# B&R Automation Studio project pneutrunk_plc (part 3)

#### Cyclic.st
```iecst
PROGRAM _CYCLIC

	TON_0(IN := kalibraciaStart, PT := T#5s0ms);

	IF buttons.klucik = FALSE THEN
		global_step		:= 0;
		step 			:= 7;
		buttons.stropBielaLED	:= FALSE;
	END_IF

	CASE step OF

		0:  // Detekcia referencnej polohy
			IF switch2 = FALSE THEN
				buttons.startLED				:= FALSE;
				switch2 						:= TRUE;
				FOR id:=0 TO 6 BY 1 DO
					modul.tlak1[id]	:= REAL_TO_INT(0);
					modul.tlak2[id]	:= REAL_TO_INT(0);
					modul.tlak3[id]	:= REAL_TO_INT(0);
					packetPos.qDesired[id*2] 	:= 0;
					packetPos.qDesired[id*2+1] 	:= 0;
					automatika.x_desired[id]	:= 0;
					automatika.y_desired[id]	:= 0;
					switch						:= FALSE;
				END_FOR

			END_IF

			IF buttons.startButton = TRUE THEN
				buttons.start	:= TRUE;
				global_step_udp	:= 0;
			END_IF

			IF buttons.start = TRUE AND buttons.centralStop = TRUE THEN
				buttons.stop					:= FALSE;
				buttons.stopLED					:= FALSE;
				buttons.stropCervenaLED			:= FALSE;
				buttons.startLED				:= TRUE;
				IF switch = FALSE THEN
					switch 						:= TRUE;
					kalibraciaStart 			:= TRUE;
					I_ON						:= TRUE;
					FOR id:=0 TO 6 BY 1 DO
						automatika.I_konstanta[id]	:= 25;
					END_FOR
					FOR id:=0 TO 6 BY 1 DO
						modul.tlak1[id]			:= REAL_TO_INT(3*32767/9);
						modul.tlak2[id]			:= REAL_TO_INT(3*32767/9);
						modul.tlak3[id]			:= REAL_TO_INT(3*32767/9);
					END_FOR
				END_IF

				IF switch = TRUE AND TON_0.Q = TRUE THEN
					switch			:= FALSE;
					kalibraciaStart	:= FALSE;
					step			:= 1;
				END_IF
			END_IF
			global_step				:= 0;
			buttons.stropBielaLED	:= TRUE;
		1:	// Vypustenie vzduchu zo vsetkych mechov, zapnutie I-regulatora
			(*
			FOR id:=0 TO 6 BY 1 DO
				modul.tlak1[id]	:= 0;
				modul.tlak2[id]	:= 0;
				modul.tlak3[id]	:= 0;
			END_FOR
			*)
			//I_ON					:= TRUE;
			switch2 				:= FALSE;
			kalibraciaStart			:= TRUE;

			step					:= 2;

		2:	// cakaj
			IF TON_0.Q = TRUE THEN
				kalibraciaStart		:= FALSE;
				step				:= 3;
			END_IF

		3:
			FOR id:=0 TO 6 BY 1 DO
				modull.nula_x[id]:= 0;
				modull.nula_y[id]:= 0;
			END_FOR

			step					:= 44;

			global_step 			:= 999;
			global_step_udp			:= 0;			// aby nahodou nemal na zaciatku gesto z predoslej udalosti

			kalibraciaStart			:= TRUE;
			(*
			FOR id:=0 TO 6 BY 1 DO
				modul.tlak1[id]	:= 0;
				modul.tlak2[id]	:= 0;
				modul.tlak3[id]	:= 0;
			END_FOR
			*)

		44:

			IF TON_0.Q = TRUE THEN
				kalibraciaStart		:= FALSE;
				step				:= 45;
				(*
				FOR id:=0 TO 6 BY 1 DO
					modull.nula_x[id]:= modul.uhol1[id]*1.0233 + 88.745;
					modull.nula_y[id]:= modul.uhol2[id];
				END_FOR
				*)
				modull.nula_x[0]:= modul.uhol1[0]*1.0233 + 88.745;
				modull.nula_x[1]:= modul.uhol1[1]*1.0228 + 88.871;
				modull.nula_x[2]:= modul.uhol1[2]*1.0235 + 90.761;
				modull.nula_x[3]:= modul.uhol1[3]*1.0254 + 88.307;
				modull.nula_x[4]:= modul.uhol1[4]*1.0216 + 90.3;
				modull.nula_x[5]:= modul.uhol1[5]*1.0039 + 87.274;
				modull.nula_x[6]:= modul.uhol1[6]*1.0065 + 87.623;

				modull.nula_y[0]:= modul.uhol2[0]*1.0275 + 89.292;
				modull.nula_y[1]:= modul.uhol2[1]*1.0079 + 89.873;
				modull.nula_y[2]:= modul.uhol2[2]*1.043 + 92.476;
				modull.nula_y[3]:= modul.uhol2[3]*1.0308 + 90.739;
				modull.nula_y[4]:= modul.uhol2[4]*1.008 + 86.877;
				modull.nula_y[5]:= modul.uhol2[5]*1.0009 + 87.856;
				modull.nula_y[6]:= modul.uhol2[6]*1.0258 + 90.567;
			END_IF
		45:
			kalibraciaStart		:= TRUE;
			step				:= 46;
		46:
			IF TON_0.Q = TRUE THEN
				kalibraciaStart	:= FALSE;
				step			:= 47;
			END_IF
		47:
			FOR id:=0 TO 6 BY 1 DO
				modul.tlak1[id]	:= 0;
				modul.tlak2[id]	:= 0;
				modul.tlak3[id]	:= 0;
			END_FOR
			step				:= 48;
			kalibraciaStart		:= TRUE;
		48:
			IF TON_0.Q = TRUE THEN
				kalibraciaStart	:= FALSE;
				step			:= 4;
			END_IF

		4:

			FOR id:=0 TO 6 BY 1 DO
			//	modull.real_uhol_x_kalibrovane[id]	:= modul.uhol1[id]*1.0233 + 88.745;
			//	modull.real_uhol_y_kalibrovane[id]	:= modul.uhol2[id];
			//	modul.uhol_XminusRef[id] 			:= modull.real_uhol_x_kalibrovane[id] - modull.nula_x[id];
			//	modul.uhol_YminusRef[id] 			:= modull.real_uhol_y_kalibrovane[id] - modull.nula_y[id];
				modul.linearReal		 			:= ref_linearny_posun;
			END_FOR

			modull.real_uhol_x_kalibrovane[0]:= modul.uhol1[0]*1.0233 + 88.745;
			modull.real_uhol_x_kalibrovane[1]:= modul.uhol1[1]*1.0228 + 88.871;
			modull.real_uhol_x_kalibrovane[2]:= modul.uhol1[2]*1.0235 + 90.761;
			modull.real_uhol_x_kalibrovane[3]:= modul.uhol1[3]*1.0254 + 88.307;
			modull.real_uhol_x_kalibrovane[4]:= modul.uhol1[4]*1.0216 + 90.3;
			modull.real_uhol_x_kalibrovane[5]:= modul.uhol1[5]*1.0039 + 87.274;
			modull.real_uhol_x_kalibrovane[6]:= modul.uhol1[6]*1.0065 + 87.623;

			modull.real_uhol_y_kalibrovane[0]:= modul.uhol2[0]*1.0275 + 89.292;
			modull.real_uhol_y_kalibrovane[1]:= modul.uhol2[1]*1.0079 + 89.873;
			modull.real_uhol_y_kalibrovane[2]:= modul.uhol2[2]*1.043 + 92.476;
			modull.real_uhol_y_kalibrovane[3]:= modul.uhol2[3]*1.0308 + 90.739;
			modull.real_uhol_y_kalibrovane[4]:= modul.uhol2[4]*1.008 + 86.877;
			modull.real_uhol_y_kalibrovane[5]:= modul.uhol2[5]*1.0009 + 87.856;
			modull.real_uhol_y_kalibrovane[6]:= modul.uhol2[6]*1.0258 + 90.567;

			IF (automatika.step_color = 1 OR automatika.step_color = 2) AND global_step = 0 THEN
				global_step			:= 999;
			END_IF

			zasobnik.ball			:= automatika.ball_up;
			zasobnik.ball_piston	:= automatika.ball_piston;
			zasobnik.ball_piston_sjf:= automatika.popcorn;
			zasobnik.levitovanie	:= automatika.levitacia;
			//modull.efektor			:= automatika.effector;
			I_konstanta_ID1			:= automatika.I_konstanta[0];
			I_konstanta_ID2			:= automatika.I_konstanta[1];
			I_konstanta_ID3			:= automatika.I_konstanta[2];
			I_konstanta_ID4			:= automatika.I_konstanta[3];
			I_konstanta_ID5			:= automatika.I_konstanta[4];
			I_konstanta_ID6			:= automatika.I_konstanta[5];
			I_konstanta_ID7			:= automatika.I_konstanta[6];

			IF buttons.stop = TRUE THEN
				buttons.start		:= FALSE;
				buttons.startLED	:= FALSE;
				buttons.stopLED		:= TRUE;
				global_step			:= 7;
			END_IF

			IF buttons.start = TRUE AND buttons.centralStop = TRUE THEN
				IF automatika.automatic = TRUE THEN
					IF automatika.holdPosition = FALSE THEN
						FOR id:=0 TO 6 BY 1 DO
							modull.pozadovany_uhol_y[id]	:=  packetPos.qDesired[id*2];
							modull.pozadovany_uhol_x[id]	:= -packetPos.qDesired[id*2+1];
						END_FOR
						modull.pozadovanyLinear				:= packetPos.qDesired[14]*7/25 + 23;
					END_IF
				ELSE
					FOR id:=0 TO 6 BY 1 DO
						modull.pozadovany_uhol_x[id]	:= automatika.x_desired[id];
						modull.pozadovany_uhol_y[id] 	:= automatika.y_desired[id];
					END_FOR
					modull.pozadovanyLinear				:= automatika.linear;
				END_IF

				// Joint limits
				FOR id:=0 TO 6 BY 1 DO
					IF modull.pozadovany_uhol_x[id] >= maxUhol THEN
						modull.pozadovany_uhol_x[id]	:= maxUhol;
					ELSIF modull.pozadovany_uhol_x[id] <= - maxUhol THEN
						modull.pozadovany_uhol_x[id] := -maxUhol;
					END_IF

					IF modull.pozadovany_uhol_y[id] >= maxUhol THEN
						modull.pozadovany_uhol_y[id]	:= maxUhol;
					ELSIF modull.pozadovany_uhol_y[id] <= - maxUhol THEN
						modull.pozadovany_uhol_y[id] := -maxUhol;
					END_IF

				END_FOR

				ref_alfa_x_ID1:= modull.pozadovany_uhol_x[0];
				ref_alfa_y_ID1:= modull.pozadovany_uhol_y[0];
				ref_alfa_x_ID2:= modull.pozadovany_uhol_x[1];
				ref_alfa_y_ID2:= modull.pozadovany_uhol_y[1];
				ref_alfa_x_ID3:= modull.pozadovany_uhol_x[2];
				ref_alfa_y_ID3:= modull.pozadovany_uhol_y[2];
				ref_alfa_x_ID4:= modull.pozadovany_uhol_x[3];
				ref_alfa_y_ID4:= modull.pozadovany_uhol_y[3];
				ref_alfa_x_ID5:= modull.pozadovany_uhol_x[4];
				ref_alfa_y_ID5:= modull.pozadovany_uhol_y[4];
				ref_alfa_x_ID6:= modull.pozadovany_uhol_x[5];
				ref_alfa_y_ID6:= modull.pozadovany_uhol_y[5];
				ref_alfa_x_ID7:= modull.pozadovany_uhol_x[6];
				ref_alfa_y_ID7:= modull.pozadovany_uhol_y[6];

				// Obmedzenie pre linearny posun (ak je hodnota nad 30 regulator sa sprava divne, nechce sa vypnut)
				IF modull.pozadovanyLinear >30 THEN
					ref_linearny_posun	:= 30;
				ELSIF modull.pozadovanyLinear <23 THEN
					ref_linearny_posun	:= 23;
				ELSE
					ref_linearny_posun	:= modull.pozadovanyLinear;
				END_IF

				(*
				act_alfa_x_ID1:= modull.real_uhol_x_kalibrovane[0] - modull.nula_x[0];
				act_alfa_y_ID1:= modull.real_uhol_y_kalibrovane[0] - modull.nula_y[0];
				act_alfa_x_ID2:= modull.real_uhol_x_kalibrovane[1] - modull.nula_x[1];
				act_alfa_y_ID2:= modull.real_uhol_y_kalibrovane[1] - modull.nula_y[1];
				act_alfa_x_ID3:= modull.real_uhol_x_kalibrovane[2] - modull.nula_x[2];
				act_alfa_y_ID3:= modull.real_uhol_y_kalibrovane[2] - modull.nula_y[2];
				act_alfa_x_ID4:= modull.real_uhol_x_kalibrovane[3] - modull.nula_x[3];
				act_alfa_y_ID4:= modull.real_uhol_y_kalibrovane[3] - modull.nula_y[3];
				act_alfa_x_ID5:= modull.real_uhol_x_kalibrovane[4] - modull.nula_x[4];
				act_alfa_y_ID5:= modull.real_uhol_y_kalibrovane[4] - modull.nula_y[4];
				act_alfa_x_ID6:= modull.real_uhol_x_kalibrovane[5] - modull.nula_x[5];
				act_alfa_y_ID6:= modull.real_uhol_y_kalibrovane[5] - modull.nula_y[5];
				act_alfa_x_ID7:= modull.real_uhol_x_kalibrovane[6] - modull.nula_x[6];
				act_alfa_y_ID7:= modull.real_uhol_y_kalibrovane[6] - modull.nula_y[6];
				*)
				(*
				act_alfa_x_ID1:= modull.real_uhol_x_kalibrovane[0] - modull.nula_x[0];
				act_alfa_y_ID1:= modull.real_uhol_y_kalibrovane[0] - modull.nula_y[0];
				act_alfa_x_ID2:= modull.real_uhol_x_kalibrovane[1] - modull.nula_x[1];
				act_alfa_y_ID2:= modull.real_uhol_y_kalibrovane[1] - modull.nula_y[1];
				act_alfa_x_ID3:= modull.real_uhol_x_kalibrovane[2] - modull.nula_x[2];
				act_alfa_y_ID3:= modull.real_uhol_y_kalibrovane[2] - modull.nula_y[2];
				act_alfa_x_ID4:= modull.real_uhol_x_kalibrovane[3] - modull.nula_x[3];
				act_alfa_y_ID4:= modull.real_uhol_y_kalibrovane[3] - modull.nula_y[3];
				act_alfa_x_ID5:= modull.real_uhol_x_kalibrovane[4] - modull.nula_x[4];
				act_alfa_y_ID5:= modull.real_uhol_y_kalibrovane[4] - modull.nula_y[4];
				act_alfa_x_ID6:= modull.real_uhol_x_kalibrovane[5] - modull.nula_x[5];
				act_alfa_y_ID6:= modull.real_uhol_y_kalibrovane[5] - modull.nula_y[5];
				act_alfa_x_ID7:= modull.real_uhol_x_kalibrovane[6] - modull.nula_x[6];
				act_alfa_y_ID7:= modull.real_uhol_y_kalibrovane[6] - modull.nula_y[6];
				*)
				// Pre experiment 2
				uhly.ref_alfa_x[0]	:= act_alfa_x_ID1;
				uhly.ref_alfa_y[0]	:= act_alfa_y_ID1;
				uhly.ref_alfa_x[1]	:= act_alfa_x_ID2;
				uhly.ref_alfa_y[1]	:= act_alfa_y_ID2;
				uhly.ref_alfa_x[2]	:= act_alfa_x_ID3;
				uhly.ref_alfa_y[2]	:= act_alfa_y_ID3;
				uhly.ref_alfa_x[3]	:= act_alfa_x_ID4;
				uhly.ref_alfa_y[3]	:= act_alfa_y_ID4;
				uhly.ref_alfa_x[4]	:= act_alfa_x_ID5;
				uhly.ref_alfa_y[4]	:= act_alfa_y_ID5;
				uhly.ref_alfa_x[5]	:= act_alfa_x_ID6;
				uhly.ref_alfa_y[5]	:= act_alfa_y_ID6;
				uhly.ref_alfa_x[6]	:= act_alfa_x_ID7;
				uhly.ref_alfa_y[6]	:= act_alfa_y_ID7;

				IF automatika.repeatability = FALSE THEN

					// Nastavenie tlakov podla regulacie
					// ID1
					id:=0;
					modul.tlak1[id] := REAL_TO_INT(Blue_tab_ID1*32767/9);
					modul.tlak2[id] := REAL_TO_INT(Green_tab_ID1*32767/9);
					modul.tlak3[id] := REAL_TO_INT(Yellow_tab_ID1*32767/9);

					// ID2
					id:=1;
					modul.tlak1[id] := REAL_TO_INT(Blue_tab_ID2*32767/9);
					modul.tlak2[id] := REAL_TO_INT(Green_tab_ID2*32767/9);
					modul.tlak3[id] := REAL_TO_INT(Yellow_tab_ID2*32767/9);

					// ID3
					id:=2;
					modul.tlak1[id] := REAL_TO_INT(Blue_tab_ID3*32767/9);
					modul.tlak2[id] := REAL_TO_INT(Green_tab_ID3*32767/9);
					modul.tlak3[id] := REAL_TO_INT(Yellow_tab_ID3*32767/9);

					// ID4
					id:=3;
					modul.tlak1[id] := REAL_TO_INT(Blue_tab_ID4*32767/9);
					modul.tlak2[id] := REAL_TO_INT(Green_tab_ID4*32767/9);
					modul.tlak3[id] := REAL_TO_INT(Yellow_tab_ID4*32767/9);

					// ID5
					id:=4;
					modul.tlak1[id] := REAL_TO_INT(Blue_tab_ID5*32767/9);
					modul.tlak2[id] := REAL_TO_INT(Green_tab_ID5*32767/9);
					modul.tlak3[id] := REAL_TO_INT(Yellow_tab_ID5*32767/9);

					// ID6
					id:=5;
					modul.tlak1[id] := REAL_TO_INT(Blue_tab_ID6*32767/9);
					modul.tlak2[id] := REAL_TO_INT(Green_tab_ID6*32767/9);
					modul.tlak3[id] := REAL_TO_INT(Yellow_tab_ID6*32767/9);

					// ID7
					id:=6;
					modul.tlak3[id] := REAL_TO_INT(Blue_tab_ID7*32767/9);
					modul.tlak1[id] := REAL_TO_INT(Green_tab_ID7*32767/9);
					modul.tlak2[id] := REAL_TO_INT(Yellow_tab_ID7*32767/9);

					//lin_modul
					modul.tlakLinear:= REAL_TO_INT(lin_pressure*32767/9);
				ELSE
					IF automatika.continuum = TRUE THEN

					ELSE

						FOR id:= 0 TO 5 BY 1 DO
							modul.tlak1[id] := automatika.desiredPressure1[id];
							modul.tlak2[id] := automatika.desiredPressure2[id];
							modul.tlak3[id] := automatika.desiredPressure3[id];
						END_FOR
						modul.tlakLinear	:= automatika.desiredPressureLinear;
					END_IF

				END_IF

			ELSIF buttons.centralStop = FALSE OR buttons.start = FALSE THEN
				buttons.start			:= FALSE;
				switch					:= FALSE;
				switch2					:= FALSE;
				I_ON					:= FALSE;
				kalibraciaStart			:= FALSE;
				step					:= 0;
				global_step_udp			:= 0;
				global_step				:= 0;
				step_repeatability		:= 0;
				automatika.repeatability:= FALSE;
				automatika.casovac		:= FALSE;
				automatika.ball_piston	:= FALSE;
				automatika.ball_up		:= FALSE;
				automatika.levitacia	:= FALSE;
				zasobnik.levitovanie	:= FALSE;
				zasobnik.ball_piston_sjf:= FALSE;
				automatika.popcorn		:= FALSE;
				automatika.casovac_uchopenie:= FALSE;
				automatika.effector		:= FALSE;
				automatika.holdPosition	:= FALSE;
				automatika.automatic	:= FALSE;
				act_alfa_x_ID1:= 0;
				act_alfa_y_ID1:= 0;
				act_alfa_x_ID2:= 0;
				act_alfa_y_ID2:= 0;
				act_alfa_x_ID3:= 0;
				act_alfa_y_ID3:= 0;
				act_alfa_x_ID4:= 0;
				act_alfa_y_ID4:= 0;
				act_alfa_x_ID5:= 0;
				act_alfa_y_ID5:= 0;
				act_alfa_x_ID6:= 0;
				act_alfa_y_ID6:= 0;
				act_alfa_x_ID7:= 0;
				act_alfa_y_ID7:= 0;
				ref_alfa_x_ID1:= 0;
				ref_alfa_y_ID1:= 0;
				ref_alfa_x_ID2:= 0;
				ref_alfa_y_ID2:= 0;
				ref_alfa_x_ID3:= 0;
				ref_alfa_y_ID3:= 0;
				ref_alfa_x_ID4:= 0;
				ref_alfa_y_ID4:= 0;
				ref_alfa_x_ID5:= 0;
				ref_alfa_y_ID5:= 0;
				ref_alfa_x_ID6:= 0;
				ref_alfa_y_ID6:= 0;
				ref_alfa_x_ID7:= 0;
				ref_alfa_y_ID7:= 0;
				FOR i:=0 TO 6 BY 1 DO
					modul.tlak1[i] 				:= 0;
					modul.tlak2[i]				:= 0;
					modul.tlak3[i] 				:= 0;
					modull.pozadovany_uhol_y[i]	:= 0;
					modull.pozadovany_uhol_x[i]	:= 0;
					modull.real_uhol_x_kalibrovane[i]	:= 0;
					modull.real_uhol_y_kalibrovane[i] 	:= 0;
					modull.nula_x[i]			:= 0;
					modull.nula_y[i]			:= 0;
				END_FOR
				modul.tlakLinear		:= 0;
			//	modull.efektor			:= FALSE;
				modull.pozadovanyLinear	:= 23;
				zasobnik.ball			:= FALSE;
				zasobnik.ball_piston	:= FALSE;
			END_IF
		5: // kolaborativny mod - doslo k narazu, alebo stlacenie stop
			buttons.startLED			:= FALSE;
			buttons.stopLED				:= TRUE;
			IF buttons.start = TRUE THEN
				buttons.stropBielaLED	:= FALSE;
				buttons.stropCervenaLED	:= TRUE;
				buttons.start			:= FALSE;
			END_IF
			step						:= 6;
			global_step					:= 0;

		6:
			IF buttons.stop = TRUE THEN
				buttons.stopLED			:= FALSE;
				buttons.stropCervenaLED	:= FALSE;
				buttons.stropBielaLED	:= TRUE;
				step					:= 7;
			END_IF

		7:	// resetovanie vsetkeho
			buttons.start			:= FALSE;
			switch					:= FALSE;
			switch2					:= FALSE;
			I_ON					:= FALSE;
			kalibraciaStart			:= FALSE;
			step					:= 0;
			global_step_udp			:= 0;
			global_step				:= 0;
			automatika.casovac		:= FALSE;
			zasobnik.levitovanie	:= FALSE;
			zasobnik.ball_piston_sjf:= FALSE;
			automatika.ball_piston	:= FALSE;
			automatika.ball_up		:= FALSE;
			automatika.popcorn		:= FALSE;
			zasobnik.ball_piston_sjf:= FALSE;
			automatika.casovac_uchopenie:= FALSE;
			automatika.effector		:= FALSE;
			automatika.holdPosition	:= FALSE;
			automatika.automatic	:= FALSE;
			act_alfa_x_ID1:= 0;
			act_alfa_y_ID1:= 0;
			act_alfa_x_ID2:= 0;
			act_alfa_y_ID2:= 0;
			act_alfa_x_ID3:= 0;
			act_alfa_y_ID3:= 0;
			act_alfa_x_ID4:= 0;
			act_alfa_y_ID4:= 0;
			act_alfa_x_ID5:= 0;
			act_alfa_y_ID5:= 0;
			act_alfa_x_ID6:= 0;
			act_alfa_y_ID6:= 0;
			act_alfa_x_ID7:= 0;
			act_alfa_y_ID7:= 0;
			ref_alfa_x_ID1:= 0;
			ref_alfa_y_ID1:= 0;
			ref_alfa_x_ID2:= 0;
			ref_alfa_y_ID2:= 0;
			ref_alfa_x_ID3:= 0;
			ref_alfa_y_ID3:= 0;
			ref_alfa_x_ID4:= 0;
			ref_alfa_y_ID4:= 0;
			ref_alfa_x_ID5:= 0;
			ref_alfa_y_ID5:= 0;
			ref_alfa_x_ID6:= 0;
			ref_alfa_y_ID6:= 0;
			ref_alfa_x_ID7:= 0;
			ref_alfa_y_ID7:= 0;
			FOR i:=0 TO 6 BY 1 DO
				modul.tlak1[i] 				:= 0;
				modul.tlak2[i]				:= 0;
				modul.tlak3[i] 				:= 0;
				modull.pozadovany_uhol_y[i]	:= 0;
				modull.pozadovany_uhol_x[i]	:= 0;
				modull.real_uhol_x_kalibrovane[i]	:= 0;
				modull.real_uhol_y_kalibrovane[i] 	:= 0;
				modull.nula_x[i]			:= 0;
				modull.nula_y[i]			:= 0;
			END_FOR
			modul.tlakLinear		:= 0;
		//	modull.efektor			:= FALSE;
			modull.pozadovanyLinear	:= 23;
			zasobnik.ball			:= FALSE;
			zasobnik.ball_piston	:= FALSE;
			IF buttons.klucik = FALSE THEN
				step				:= 8;
				global_step			:= 0;
			ELSE
				step				:= 0;
			END_IF
		8:
			IF buttons.klucik = TRUE THEN
				step				:= 0;
				global_step			:= 0;
			ELSE
				buttons.stropBielaLED	:= FALSE;
			END_IF

	END_CASE

	IF I_ON= TRUE THEN
		RESET_ID1:= TRUE;
		RESET_ID2:= TRUE;
		RESET_ID3:= TRUE;
		RESET_ID4:= TRUE;
		RESET_ID5:= TRUE;
		RESET_ID6:= TRUE;
		RESET_ID7:= TRUE;
	ELSE
		RESET_ID1:= FALSE;
		RESET_ID2:= FALSE;
		RESET_ID3:= FALSE;
		RESET_ID4:= FALSE;
		RESET_ID5:= FALSE;
		RESET_ID6:= FALSE;
		RESET_ID7:= FALSE;
	END_IF

	I_konstanta_ID1;
	I_konstanta_ID2;
	I_konstanta_ID3;
	I_konstanta_ID4;
	I_konstanta_ID5;
	I_konstanta_ID6;
	I_konstanta_ID7;

END_PROGRAM
```

#### Init.st
```iecst
PROGRAM _INIT
//	traj_0(ssMethodType := 2, aktualny_uhol_x := 0, aktualny_uhol_y := 0, pozadovany_uhol_x := 0, pozadovany_uhol_y :=0, dlzka_pohybu := 1);

//	traj_1(ssMethodType := 2, aktualny_uhol_x := 0, aktualny_uhol_y := 0, pozadovany_uhol_x := 0, pozadovany_uhol_y :=0, dlzka_pohybu := 1);

//	uhol2zdvyh_0(ssMethodType := 2, uhol_x := 15, uhol_y := 15);

	//FF_PID_r_t_0(ssMethodType := 0, ref_alfa_x := 0, ref_alfa_y := 0, real_alfa_x := 0, real_alfa_y := 0, P_parameter := 0, reset_PID_blue := 0, D_parameter := 0, N_parameter := 0, stiffness_ff := 3, reset_PID_green := 0, reset_PID_yellow := 0, tlak3 := 0, I_parameter := 0, tlak1 := 0, tlak2 := 0);
	FOR id:=0 TO 6 BY 1 DO
		modull.poradie[id]	:= 3;
	END_FOR

	maxUhol := 18;

	modull.FF_stiffness[0]	:= 3;
	stiffness_ff:= modull.FF_stiffness[0];
	switch := FALSE;
	poradie_ID1:=3;
	poradie_ID2:=3;
	poradie_ID3:=3;
	poradie_ID4:=3;
	poradie_ID5:=3;
	poradie_ID6:=3;
	poradie_ID7:=3;

	I_konstanta_ID1:=30;
	I_konstanta_ID2:=30;
	I_konstanta_ID3:=30;
	I_konstanta_ID4:=30;
	I_konstanta_ID5:=30;
	I_konstanta_ID6:=30;
	I_konstanta_ID7:=30;

	IF buttons.klucik = TRUE THEN
		buttons.stropBielaLED	:= TRUE;
	END_IF

	buttons.stropCervenaLED	:= FALSE;

END_PROGRAM
```

### Program Logical/Source/RS485/Sender (IEC) - sending serial data

#### SenderCyclic.st
```iecst
(********************************************************************
 * COPYRIGHT -- Bernecker + Rainer
 ********************************************************************
 * Program: Sender
 * File: SenderCyclic.st
 * Author: Bernecker & Rainer
 * Created: January 25, 2010
 ********************************************************************
 * Implementation of program Sender
 ********************************************************************)

(*************init program**********************)
PROGRAM _INIT
	Sender.Commands.open_send := TRUE;												(*enable sender by default*)
	packet485.sendPacketFinal[0] := 255;
	packet485.sendPacketFinal[1] := 255;
	packet485.sendPacketFinal[2] := 1;				// ID
	packet485.sendPacketFinal[3] := 1;
	packet485.sendPacketFinal[4] := 254;
	packet485.sendPacketFinal[5] := 254;
	Sender.step					 := FRM_WAIT;
END_PROGRAM

(*************cyclic program********************)
PROGRAM _CYCLIC

	CASE Sender.step OF
		FRM_WAIT:	(*--- wait for command*)

			IF Sender.Commands.open_send = TRUE THEN								(*command for sender activation*)
				Sender.step := FRM_OPEN;
   			END_IF

			(*close will be requested in step FRM_WRITE*)

		FRM_OPEN:	(*--- open serial interface*)

			(*Parameters for FRM_xopen()*)
			Sender.FRM_xopen_0.enable := TRUE;
			Sender.FRM_xopen_0.device := ADR('IF6.ST1.IF1');										(*Devicename --> see your serial interface properties*)
			Sender.FRM_xopen_0.mode := ADR('/PHY=RS485 /BD=38400 /DB=8 /PA=N /SB=1'); 		(*Modestring --> specifies the seria operation mode*)
			Sender.FRM_xopen_0.config := ADR(Sender.xopenConfig) ;					(*Additional Parameters, optional*)

			(*Additional Parameters for FRM_xopen()*)
			Sender.xopenConfig.idle := 10;											(*Idle time between two characters*)
			Sender.xopenConfig.delimc := 0;											(*activate two delimeters*)
			Sender.xopenConfig.delim[0] := 0; 										(*CR - carridge return -> dec 13*)
			Sender.xopenConfig.delim[1] := 0; 										(*LF - line feed -> dec 10*)
			Sender.xopenConfig.tx_cnt := 3;											(*number of transmit buffers*)
			Sender.xopenConfig.rx_cnt := 3; 										(*number of receive buffers*)
			Sender.xopenConfig.tx_len := 256; 										(*length of transmit buffers*)
			Sender.xopenConfig.rx_len := 256; 										(*lenght of receive buffers*)
			Sender.xopenConfig.argc := 0;											(*activate additional options*)
			Sender.xopenConfig.argv := 0;											(*parameters for additional options (check help)*)

			Sender.FRM_xopen_0();													(*call the FRM_xopen() function*)

			IF Sender.FRM_xopen_0.status = 0 THEN
				Sender.step := FRM_GBUF;											(*Interface opend successfully --> next step*)
			ELSIF Sender.FRM_xopen_0.status = BUSY THEN
				Sender.step := FRM_OPEN;											(*operation not finished yet --> call again*)
			ELSE
				Sender.step := FRM_ERROR;											(*function returned errorcode --> check help*)
   			END_IF

		FRM_GBUF:	(*--- aquire sendbuffer for FRM_WRITE*)
			Sender.FRM_gbuf_0.enable := TRUE;
   			Sender.FRM_gbuf_0.ident := Sender.FRM_xopen_0.ident;

			Sender.FRM_gbuf_0();													(*call the FRM_gbuf() function*)

			IF Sender.FRM_gbuf_0.status = 0 THEN
				memset(Sender.FRM_gbuf_0.buffer,0,Sender.FRM_gbuf_0.buflng);		(*clear sendbuffer*)
				Sender.step := FRM_PREPARE_SENDDATA;								(*system returned a valid buffer --> next step*)
			ELSIF Sender.FRM_gbuf_0.status = BUSY THEN
				Sender.step := FRM_GBUF;											(*operation not finished yet --> call again*)
			ELSE
				Sender.step := FRM_ERROR;											(*function returned errorcode --> check help*)
   			END_IF

		FRM_PREPARE_SENDDATA: (*--- prepare senddata, copy data to sendbuffer*)

			IF packet485.id = 8 THEN
				packet485.id := 1;
			ELSE
				packet485.id := packet485.id + 1;
			END_IF
			Sender.Commands.open_send := TRUE;										(*enable sender by default*)
			packet485.sendPacketFinal[0] := 255;
			packet485.sendPacketFinal[1] := 255;
			packet485.sendPacketFinal[2] := USINT_TO_BYTE(packet485.id);
			packet485.sendPacketFinal[3] := 1;
			packet485.sendPacketFinal[4] := 254;
			packet485.sendPacketFinal[5] := 254;
			packet485.sendPacketFinal[0] := 255;

			strcpy(Sender.FRM_gbuf_0.buffer,ADR(packet485.sendPacketFinal));		(*copy senddata to sendbuffer*)
			Sender.step := FRM_WRITE;												(*--> next step*)

		FRM_WRITE:	(*--- write data to interface*)

			(*Parameters for FRM_write()*)
			Sender.FRM_write_0.enable := TRUE;
			Sender.FRM_write_0.ident := Sender.FRM_xopen_0.ident;					(*ident from FRM_xopen()*)
			Sender.FRM_write_0.buffer := Sender.FRM_gbuf_0.buffer;					(*sendbuffer*)
			Sender.FRM_write_0.buflng := strlen(ADR(packet485.sendPacketFinal));				(*net length of senddata*)

			Sender.FRM_write_0();													(*call the FRM_write() function*)

			IF Sender.FRM_write_0.status = 0 THEN
				IF Sender.Commands.close = TRUE THEN								(*requst to close the serial port*)
					Sender.Commands.open_send := FALSE;								(*disable command open_send*)
					Sender.step := FRM_CLOSE;
				ELSE
					Sender.step := FRM_GBUF;										(*writing successful --> get next sendbuffer*)
				END_IF
			ELSIF Sender.FRM_write_0.status = BUSY THEN
				Sender.step := FRM_WRITE;											(*operation not finished yet --> call again*)
			ELSE
				Sender.step := FRM_ROBUF;											(*function returned errorcode --> check help*)
   			END_IF

		FRM_ROBUF:	(*--- release sendbuffer in case of no successful write operation*)
			Sender.FRM_robuf_0.enable := TRUE;
			Sender.FRM_robuf_0.buffer := Sender.FRM_gbuf_0.buffer;					(*sendbuffer*)
			Sender.FRM_robuf_0.buflng := Sender.FRM_gbuf_0.buflng;					(*buffer length*)
			Sender.FRM_robuf_0.ident := Sender.FRM_xopen_0.ident;					(*ident open*)

			Sender.FRM_robuf_0();													(*call the FRM_robuf() function*)

			IF Sender.FRM_robuf_0.status = 0 THEN
				Sender.step := FRM_GBUF;											(*released buffer successful --> get next sendbuffer*)
			ELSIF Sender.FRM_robuf_0.status = BUSY THEN
				Sender.step := FRM_ROBUF;											(*operation not finished yet --> call again*)
			ELSE
				Sender.step := FRM_ERROR;											(*function returned errorcode --> check help*)
   			END_IF

		FRM_CLOSE:	(*--- close the interface*)
			Sender.FRM_close_0.enable := TRUE;
   			Sender.FRM_close_0.ident := Sender.FRM_xopen_0.ident;					(*ident from FRM_xopen()*)

			Sender.FRM_close_0();													(*call the FRM_close() function*)

			IF Sender.FRM_close_0.status = 0 THEN
				Sender.Commands.close := FALSE;										(*disable close command*)
				Sender.step := FRM_WAIT;											(*closed interface successfully --> wait step*)
			ELSIF Sender.FRM_close_0.status = BUSY THEN
				Sender.step := FRM_CLOSE;											(*operation not finished yet --> call again*)
			ELSE
				Sender.step := FRM_ERROR;											(*function returned errorcode --> check help*)
			END_IF

		FRM_ERROR:	(*--- error handling*)
			Sender.step := FRM_WAIT;
			//; (*not implementet yet, check help for error codes*)
 	END_CASE

END_PROGRAM
```

### Program Logical/Source/RS485/Receiver (IEC) - receiving serial data

#### ReceiverCyclic.st
```iecst
(********************************************************************
 * COPYRIGHT -- Bernecker + Rainer
 ********************************************************************
 * Program: Receiver
 * File: ReceiverCyclic.st
 * Author: Bernecker & Rainer
 * Created: January 25, 2010
 ********************************************************************
 * Implementation of program Receiver
 ********************************************************************)

(*************init program**********************)
PROGRAM _INIT
	Receiver.Commands.open_receive := TRUE;												(*enable Receiver by default*)
END_PROGRAM

(*************cyclic program********************)
PROGRAM _CYCLIC

	CASE Receiver.step OF
		FRM_WAIT:	(*--- wait for command*)

			IF Receiver.Commands.open_receive = TRUE THEN								(*command for Receiver activation*)
				Receiver.step := FRM_OPEN;
   			END_IF

			(*close will be requested in step FRM_RBUF*)

		FRM_OPEN:	(*--- open serial interface*)

			(*Parameters for FRM_xopen()*)
			Receiver.FRM_xopen_0.enable := TRUE;
			Receiver.FRM_xopen_0.device := ADR('IF6.ST1.IF1');							(*Devicename --> see your serial interface properties*)
			Receiver.FRM_xopen_0.mode := ADR('/PHY=RS485 /BD=38400 /DB=8 /PA=N /SB=1'); (*Modestring --> specifies the seria operation mode*)
			Receiver.FRM_xopen_0.config := ADR(Receiver.xopenConfig) ;					(*Additional Parameters, optional*)

			(*Additional Parameters for FRM_xopen()*)
			Receiver.xopenConfig.idle := 10;											(*Idle time between two characters*)
			Receiver.xopenConfig.delimc := 0;											(*activate two delimeters*)
			Receiver.xopenConfig.delim[0] := 0; 										(*e.g. CR - carridge return -> dec 13*)
			Receiver.xopenConfig.delim[1] := 0; 										(*e.g. LF - line feed -> dec 10*)
			Receiver.xopenConfig.tx_cnt := 3;											(*number of transmit buffers*)
			Receiver.xopenConfig.rx_cnt := 3; 											(*number of receive buffers*)
			Receiver.xopenConfig.tx_len := 256; 										(*length of transmit buffers*)
			Receiver.xopenConfig.rx_len := 256; 										(*lenght of receive buffers*)
			Receiver.xopenConfig.argc := 0;												(*activate additional options*)
			Receiver.xopenConfig.argv := 0;												(*parameters for additional options (check help)*)

			Receiver.FRM_xopen_0();														(*call the FRM_xopen() function*)

			IF Receiver.FRM_xopen_0.status = 0 THEN
				Receiver.step := FRM_READ;												(*Interface opend successfully --> next step*)
			ELSIF Receiver.FRM_xopen_0.status = BUSY THEN
				Receiver.step := FRM_OPEN;												(*operation not finished yet --> call again*)
			ELSE
				Receiver.step := FRM_ERROR;												(*function returned errorcode --> check help*)
   			END_IF

		FRM_READ:	(*--- read data from serial interface*)
			Receiver.FRM_read_0.enable := TRUE;
   			Receiver.FRM_read_0.ident := Receiver.FRM_xopen_0.ident;

			Receiver.FRM_read_0();														(*call the FRM_read() function*)

			IF Receiver.FRM_read_0.status = 0 THEN
				Receiver.step := FRM_COPY_RD_DATA;										(*system returned a valid data --> next step*)
			ELSIF Receiver.FRM_read_0.status = frmERR_NOINPUT THEN
				Receiver.step := FRM_READ;												(*no data available --> call again*)
			ELSIF Receiver.FRM_read_0.status = frmERR_INPUTERROR THEN
				Receiver.step := FRM_RBUF;												(*received Frame with defective characters, skip data*)
			ELSE
				Receiver.step := FRM_ERROR;												(*function returned errorcode --> check help*)
   			END_IF

		FRM_COPY_RD_DATA: (*--- copy data out of the receive buffer*)
			(*
			FOR i:=0 TO 8 BY 1 DO
				packet485.packet[i] := Receiver.receive_data[i];
			END_FOR
			*)
			memset(ADR(Receiver.receive_data),0,SIZEOF(Receiver.receive_data));			(*clear read_data buffer*)
			memcpy(ADR(Receiver.receive_data),Receiver.FRM_read_0.buffer,Receiver.FRM_read_0.buflng);     (*copy and evaluate read data*)

			IF(Receiver.receive_data[0] = 255)THEN
				IF(Receiver.receive_data[1] = 255)THEN
					IF(Receiver.receive_data[9] = 254)THEN
						IF(Receiver.receive_data[10] = 254)THEN
							IF(Receiver.receive_data[2] = 1)THEN
								modul.uholINT1 := BYTE_TO_INT(Receiver.receive_data[5]);
								modul.uholINT1 := SHL(modul.uholINT1,8);
								modul.uholINT1  := modul.uholINT1  + BYTE_TO_INT(Receiver.receive_data[6]);
								modul.uhol1[0] := INT_TO_REAL(modul.uholINT1);
								modul.uhol1[0] := modul.uhol1[0]*260/1024 - 130;
								modul.uholINT2 := BYTE_TO_INT(Receiver.receive_data[7]);
								modul.uholINT2 := SHL(modul.uholINT2,8);
								modul.uholINT2  := modul.uholINT2  + BYTE_TO_INT(Receiver.receive_data[8]);
								modul.uhol2[0] := INT_TO_REAL(modul.uholINT2);
								modul.uhol2[0] := modul.uhol2[0]*260/1024 - 130;
							ELSIF(Receiver.receive_data[2] = 2)THEN
								modul.uholINT1 := BYTE_TO_INT(Receiver.receive_data[5]);
								modul.uholINT1 := SHL(modul.uholINT1,8);
								modul.uholINT1  := modul.uholINT1  + BYTE_TO_INT(Receiver.receive_data[6]);
								modul.uhol1[1] := INT_TO_REAL(modul.uholINT1);
								modul.uhol1[1] := modul.uhol1[1]*260/1024 - 130;
								modul.uholINT2 := BYTE_TO_INT(Receiver.receive_data[7]);
								modul.uholINT2 := SHL(modul.uholINT2,8);
								modul.uholINT2  := modul.uholINT2  + BYTE_TO_INT(Receiver.receive_data[8]);
								modul.uhol2[1] := INT_TO_REAL(modul.uholINT2);
								modul.uhol2[1] := modul.uhol2[1]*260/1024 - 130;
							ELSIF(Receiver.receive_data[2] = 3)THEN
								modul.uholINT1 := BYTE_TO_INT(Receiver.receive_data[5]);
								modul.uholINT1 := SHL(modul.uholINT1,8);
								modul.uholINT1  := modul.uholINT1  + BYTE_TO_INT(Receiver.receive_data[6]);
								modul.uhol1[2] := INT_TO_REAL(modul.uholINT1);
								modul.uhol1[2] := modul.uhol1[2]*260/1024 - 130;
								modul.uholINT2 := BYTE_TO_INT(Receiver.receive_data[7]);
								modul.uholINT2 := SHL(modul.uholINT2,8);
								modul.uholINT2  := modul.uholINT2  + BYTE_TO_INT(Receiver.receive_data[8]);
								modul.uhol2[2] := INT_TO_REAL(modul.uholINT2);
								modul.uhol2[2] := modul.uhol2[2]*260/1024 - 130;
								IF Receiver.receive_data[4] = 3 OR Receiver.receive_data[4] > 15 THEN
									modul.naraz[2]	:= TRUE;
								ELSE
									modul.naraz[2]	:= FALSE;
								END_IF
							ELSIF(Receiver.receive_data[2] = 4)THEN
								modul.uholINT1 := BYTE_TO_INT(Receiver.receive_data[5]);
								modul.uholINT1 := SHL(modul.uholINT1,8);
								modul.uholINT1  := modul.uholINT1  + BYTE_TO_INT(Receiver.receive_data[6]);
								modul.uhol1[3] := INT_TO_REAL(modul.uholINT1);
								modul.uhol1[3] := modul.uhol1[3]*260/1024 - 130;
								modul.uholINT2 := BYTE_TO_INT(Receiver.receive_data[7]);
								modul.uholINT2 := SHL(modul.uholINT2,8);
								modul.uholINT2  := modul.uholINT2  + BYTE_TO_INT(Receiver.receive_data[8]);
								modul.uhol2[3] := INT_TO_REAL(modul.uholINT2);
								modul.uhol2[3] := modul.uhol2[3]*260/1024 - 130;
								IF Receiver.receive_data[4] = 3 OR Receiver.receive_data[4] > 15 THEN
									modul.naraz[3]	:= TRUE;
								ELSE
									modul.naraz[3]	:= FALSE;
								END_IF
							ELSIF(Receiver.receive_data[2] = 5)THEN
								modul.uholINT1 := BYTE_TO_INT(Receiver.receive_data[5]);
								modul.uholINT1 := SHL(modul.uholINT1,8);
								modul.uholINT1  := modul.uholINT1  + BYTE_TO_INT(Receiver.receive_data[6]);
								modul.uhol1[4] := INT_TO_REAL(modul.uholINT1);
								modul.uhol1[4] := modul.uhol1[4]*260/1024 - 130;
								modul.uholINT2 := BYTE_TO_INT(Receiver.receive_data[7]);
								modul.uholINT2 := SHL(modul.uholINT2,8);
								modul.uholINT2  := modul.uholINT2  + BYTE_TO_INT(Receiver.receive_data[8]);
								modul.uhol2[4] := INT_TO_REAL(modul.uholINT2);
								modul.uhol2[4] := modul.uhol2[4]*260/1024 - 130;
								IF Receiver.receive_data[4] = 3 OR Receiver.receive_data[4] > 15  THEN
									modul.naraz[4]	:= TRUE;
								ELSE
									modul.naraz[4]	:= FALSE;
								END_IF
							ELSIF(Receiver.receive_data[2] = 6)THEN
								modul.uholINT1 := BYTE_TO_INT(Receiver.receive_data[5]);
								modul.uholINT1 := SHL(modul.uholINT1,8);
								modul.uholINT1  := modul.uholINT1  + BYTE_TO_INT(Receiver.receive_data[6]);
								modul.uhol1[5] := INT_TO_REAL(modul.uholINT1);
								modul.uhol1[5] := modul.uhol1[5]*260/1024 - 130;
								modul.uholINT2 := BYTE_TO_INT(Receiver.receive_data[7]);
								modul.uholINT2 := SHL(modul.uholINT2,8);
								modul.uholINT2  := modul.uholINT2  + BYTE_TO_INT(Receiver.receive_data[8]);
								modul.uhol2[5] := INT_TO_REAL(modul.uholINT2);
								modul.uhol2[5] := modul.uhol2[5]*260/1024 - 130;
								IF Receiver.receive_data[4] = 3 OR Receiver.receive_data[4] > 15 THEN
									modul.naraz[5]	:= TRUE;
								ELSE
									modul.naraz[5]	:= FALSE;
								END_IF
							ELSIF(Receiver.receive_data[2] = 7)THEN
								modul.uholINT1 := BYTE_TO_INT(Receiver.receive_data[5]);
								modul.uholINT1 := SHL(modul.uholINT1,8);
								modul.uholINT1  := modul.uholINT1  + BYTE_TO_INT(Receiver.receive_data[6]);
								modul.uhol1[6] := INT_TO_REAL(modul.uholINT1);
								modul.uhol1[6] := modul.uhol1[6]*260/1024 - 130;
								modul.uholINT2 := BYTE_TO_INT(Receiver.receive_data[7]);
								modul.uholINT2 := SHL(modul.uholINT2,8);
								modul.uholINT2  := modul.uholINT2  + BYTE_TO_INT(Receiver.receive_data[8]);
								modul.uhol2[6] := INT_TO_REAL(modul.uholINT2);
								modul.uhol2[6] := modul.uhol2[6]*260/1024 - 130;
								IF Receiver.receive_data[4] = 1 OR Receiver.receive_data[4] = 2 OR Receiver.receive_data[4] > 15  THEN //lebo dve moduly su zapojene do jednej dosky
									modul.naraz[6]	:= TRUE;
								ELSE
									modul.naraz[6]	:= FALSE;
								END_IF
							ELSIF(Receiver.receive_data[2] = 8)THEN
								IF Receiver.receive_data[4] = 3 OR Receiver.receive_data[4] > 15 THEN
									modul.naraz[7]	:= TRUE;
								ELSE
									modul.naraz[7]	:= FALSE;
								END_IF
							END_IF
						END_IF
					END_IF
				END_IF
			END_IF

			Receiver.step := FRM_RBUF;													(*release read buffer*)

		FRM_RBUF:	(*--- release readbuffer*)

			(*Parameters for FRM_rbuf()*)
			Receiver.FRM_rbuf_0.enable := TRUE;
			Receiver.FRM_rbuf_0.ident := Receiver.FRM_xopen_0.ident;					(*ident from FRM_xopen()*)
			Receiver.FRM_rbuf_0.buffer := Receiver.FRM_read_0.buffer;					(*read buffer*)
			Receiver.FRM_rbuf_0.buflng := Receiver.FRM_read_0.buflng;					(*length of sendbuffer*)

			Receiver.FRM_rbuf_0();														(*call the FRM_rbuf() function*)

			IF Receiver.FRM_rbuf_0.status = 0 THEN
				IF Receiver.Commands.close = TRUE THEN
					Receiver.Commands.open_receive := FALSE;								(*disable command open_send*)
					Receiver.step := FRM_CLOSE;											(*request to close serial port*)
				ELSE
					Receiver.step := FRM_READ;											(*read again*)
				END_IF
			ELSIF Receiver.FRM_rbuf_0.status = BUSY THEN
				Receiver.step := FRM_RBUF;												(*operation not finished yet --> call again*)
			ELSIF Receiver.FRM_rbuf_0.status = frmERR_INVALIDBUFFER THEN
				Receiver.step := FRM_READ;												(*buffer is invalid --> read again*)
			ELSE
				Receiver.step := FRM_ERROR;												(*function returned errorcode --> check help*)
   			END_IF

		FRM_CLOSE:	(*--- close the interface*)
			Receiver.FRM_close_0.enable := TRUE;
   			Receiver.FRM_close_0.ident := Receiver.FRM_xopen_0.ident;					(*ident from FRM_xopen()*)

			Receiver.FRM_close_0();														(*call the FRM_close() function*)

			IF Receiver.FRM_close_0.status = 0 THEN
				Receiver.Commands.close := FALSE;										(*disable close command*)
				Receiver.step := FRM_WAIT;												(*closed interface successfully --> wait step*)
			ELSIF Receiver.FRM_close_0.status = BUSY THEN
				Receiver.step := FRM_CLOSE;												(*operation not finished yet --> call again*)
			ELSE
				Receiver.step := FRM_ERROR;												(*function returned errorcode --> check help*)
			END_IF

		FRM_ERROR:	(*--- error handling*)
			; (*not implementet yet, check help for error codes*)
 	END_CASE

END_PROGRAM
```

### Program Logical/Source/Testing (IEC)

#### Cyclic.st
```iecst
PROGRAM _CYCLIC

	IF i >= 30000 THEN
		i := 0;
	ELSE
		i := i + 100;
	END_IF

	modul.tlak1[0] := i;

END_PROGRAM
```

### Program Logical/Source/Experiments/Continuum

#### Variables.var
```iecst
VAR
	pressure : tlak;
	id : INT;
END_VAR
```

#### Cyclic.st
```iecst
PROGRAM _CYCLIC
	automatika.continuum	:= TRUE;
	FOR id:=0 TO 5 BY 1 DO
		modul.tlak1[id]	:= REAL_TO_INT(pressure.p1*32767/9);
		modul.tlak2[id]	:= REAL_TO_INT(pressure.p2*32767/9);
		modul.tlak3[id]	:= REAL_TO_INT(pressure.p3*32767/9);
	END_FOR
	modul.tlak2[6]	:= REAL_TO_INT(pressure.p3*32767/9);
	modul.tlak3[6]	:= REAL_TO_INT(pressure.p2*32767/9);
	modul.tlak1[6]	:= REAL_TO_INT(pressure.p1*32767/9);

END_PROGRAM
```

### Program Logical/Source/Experiments/HandControl

#### Cyclic.st
```iecst
PROGRAM _CYCLIC

	FOR id:=0 TO 6 BY 1 DO
		automatika.x_desired[id]	:= (uhly.ref_alfa_x[id]);
		automatika.y_desired[id]	:= (uhly.ref_alfa_y[id]);
	END_FOR

END_PROGRAM
```

### Program Logical/Source/Experiments/Repeatability

#### Variables.var
```iecst
VAR
	casovac_start : BOOL;
	TON_0 : TON;
	i : INT;
	TON_1 : TON;
	pauza : BOOL;
	TON_2 : TON;
	kameraBool : BOOL;
END_VAR
```

#### Cyclic.st
```iecst
PROGRAM _CYCLIC

	TON_0(IN := casovac_start, PT := INT_TO_TIME(automatika.cas));
	TON_1(IN := pauza, PT := T#10s0ms);
	TON_2(IN := kameraBool, PT := T#1s0ms);

	IF step = 4 THEN

		CASE automatika.step_repeatability OF
			0:
				casovac_start					:= TRUE;
				automatika.step_repeatability	:= 1;
				automatika.repeatability		:= TRUE;
				automatika.cas					:= 5000;

			1:	// Point A
				automatika.desiredPressure1[0]:= TIME_TO_INT(TON_0.ET)*1669/((automatika.cas));
				automatika.desiredPressure1[1]:= TIME_TO_INT(TON_0.ET)*3013/((automatika.cas));
				automatika.desiredPressure1[2]:= TIME_TO_INT(TON_0.ET)*(-4146)/((automatika.cas));
				automatika.desiredPressure1[3]:= TIME_TO_INT(TON_0.ET)*(-8424)/((automatika.cas));
				automatika.desiredPressure1[4]:= TIME_TO_INT(TON_0.ET)*335/((automatika.cas));
				automatika.desiredPressure1[5]:= TIME_TO_INT(TON_0.ET)*2453/((automatika.cas));
				automatika.desiredPressure1[6]:= TIME_TO_INT(TON_0.ET)*6053/((automatika.cas));

				automatika.desiredPressure2[0]:= TIME_TO_INT(TON_0.ET)*6958/((automatika.cas));
				automatika.desiredPressure2[1]:= TIME_TO_INT(TON_0.ET)*4381/((automatika.cas));
				automatika.desiredPressure2[2]:= TIME_TO_INT(TON_0.ET)*12008/((automatika.cas));
				automatika.desiredPressure2[3]:= TIME_TO_INT(TON_0.ET)*13312/((automatika.cas));
				automatika.desiredPressure2[4]:= TIME_TO_INT(TON_0.ET)*8361/((automatika.cas));
				automatika.desiredPressure2[5]:= TIME_TO_INT(TON_0.ET)*6761/((automatika.cas));
				automatika.desiredPressure2[6]:= TIME_TO_INT(TON_0.ET)*3567/((automatika.cas));

				automatika.desiredPressure3[0]:= TIME_TO_INT(TON_0.ET)*4006/((automatika.cas));
				automatika.desiredPressure3[1]:= TIME_TO_INT(TON_0.ET)*5379/((automatika.cas));
				automatika.desiredPressure3[2]:= TIME_TO_INT(TON_0.ET)*5605/((automatika.cas));
				automatika.desiredPressure3[3]:= TIME_TO_INT(TON_0.ET)*3560/((automatika.cas));
				automatika.desiredPressure3[4]:= TIME_TO_INT(TON_0.ET)*3900/((automatika.cas));
				automatika.desiredPressure3[5]:= TIME_TO_INT(TON_0.ET)*3205/((automatika.cas));
				automatika.desiredPressure3[6]:= TIME_TO_INT(TON_0.ET)*2770/((automatika.cas));

				automatika.desiredPressureLinear := TIME_TO_INT(TON_0.ET)*10800/((automatika.cas));

				IF TON_0.Q = TRUE THEN
					casovac_start					:= FALSE;
					automatika.step_repeatability	:= 2;
					FOR i:=0 TO 6 BY 1 DO
						automatika.desiredPressure1_previous[i]		:= automatika.desiredPressure1[i];
						automatika.desiredPressure2_previous[i]		:= automatika.desiredPressure2[i];
						automatika.desiredPressure3_previous[i]		:= automatika.desiredPressure3[i];
					END_FOR
				END_IF

			2:	// Pause
				pauza								:= TRUE;
				automatika.step_repeatability		:= 3;
			3:
				IF TON_1.Q = TRUE THEN
					pauza							:= FALSE;
					automatika.step_repeatability	:= 44;
					casovac_start					:= TRUE;
					kameraBool						:= TRUE;
				END_IF
			44:
				IF TON_2.Q = TRUE THEN
					kameraBool						:= FALSE;
					automatika.step_repeatability	:= 4;
				END_IF

			4:	// Point B
				automatika.desiredPressure1[0]:= (automatika.desiredPressure1_previous[0]*(automatika.cas - TIME_TO_INT(TON_0.ET))/automatika.cas) + TIME_TO_INT(TON_0.ET)*(5403)/(automatika.cas);
				automatika.desiredPressure1[1]:= (automatika.desiredPressure1_previous[1]*(automatika.cas - TIME_TO_INT(TON_0.ET))/automatika.cas) + TIME_TO_INT(TON_0.ET)*(5622)/(automatika.cas);
				automatika.desiredPressure1[2]:= (automatika.desiredPressure1_previous[2]*(automatika.cas - TIME_TO_INT(TON_0.ET))/automatika.cas) + TIME_TO_INT(TON_0.ET)*(7940)/(automatika.cas);
				automatika.desiredPressure1[3]:= (automatika.desiredPressure1_previous[3]*(automatika.cas - TIME_TO_INT(TON_0.ET))/automatika.cas) + TIME_TO_INT(TON_0.ET)*(6420)/(automatika.cas);
				automatika.desiredPressure1[4]:= (automatika.desiredPressure1_previous[4]*(automatika.cas - TIME_TO_INT(TON_0.ET))/automatika.cas) + TIME_TO_INT(TON_0.ET)*(8355)/(automatika.cas);
				automatika.desiredPressure1[5]:= (automatika.desiredPressure1_previous[5]*(automatika.cas - TIME_TO_INT(TON_0.ET))/automatika.cas) + TIME_TO_INT(TON_0.ET)*(6516)/(automatika.cas);
				automatika.desiredPressure1[6]:= (automatika.desiredPressure1_previous[6]*(automatika.cas - TIME_TO_INT(TON_0.ET))/automatika.cas) + TIME_TO_INT(TON_0.ET)*(565)/(automatika.cas);

				automatika.desiredPressure2[0]:= (automatika.desiredPressure2_previous[0]*(automatika.cas - TIME_TO_INT(TON_0.ET))/automatika.cas) + TIME_TO_INT(TON_0.ET)*(1406)/(automatika.cas);
				automatika.desiredPressure2[1]:= (automatika.desiredPressure2_previous[1]*(automatika.cas - TIME_TO_INT(TON_0.ET))/automatika.cas) + TIME_TO_INT(TON_0.ET)*(2287)/(automatika.cas);
				automatika.desiredPressure2[2]:= (automatika.desiredPressure2_previous[2]*(automatika.cas - TIME_TO_INT(TON_0.ET))/automatika.cas) + TIME_TO_INT(TON_0.ET)*(271)/(automatika.cas);
				automatika.desiredPressure2[3]:= (automatika.desiredPressure2_previous[3]*(automatika.cas - TIME_TO_INT(TON_0.ET))/automatika.cas) + TIME_TO_INT(TON_0.ET)*(2520)/(automatika.cas);
				automatika.desiredPressure2[4]:= (automatika.desiredPressure2_previous[4]*(automatika.cas - TIME_TO_INT(TON_0.ET))/automatika.cas) + TIME_TO_INT(TON_0.ET)*(829)/(automatika.cas);
				automatika.desiredPressure2[5]:= (automatika.desiredPressure2_previous[5]*(automatika.cas - TIME_TO_INT(TON_0.ET))/automatika.cas) + TIME_TO_INT(TON_0.ET)*(1928)/(automatika.cas);
				automatika.desiredPressure2[6]:= (automatika.desiredPressure2_previous[6]*(automatika.cas - TIME_TO_INT(TON_0.ET))/automatika.cas) + TIME_TO_INT(TON_0.ET)*(4860)/(automatika.cas);

				automatika.desiredPressure3[0]:= (automatika.desiredPressure3_previous[0]*(automatika.cas - TIME_TO_INT(TON_0.ET))/automatika.cas) + TIME_TO_INT(TON_0.ET)*(5933)/(automatika.cas);
				automatika.desiredPressure3[1]:= (automatika.desiredPressure3_previous[1]*(automatika.cas - TIME_TO_INT(TON_0.ET))/automatika.cas) + TIME_TO_INT(TON_0.ET)*(4731)/(automatika.cas);
				automatika.desiredPressure3[2]:= (automatika.desiredPressure3_previous[2]*(automatika.cas - TIME_TO_INT(TON_0.ET))/automatika.cas) + TIME_TO_INT(TON_0.ET)*(4820)/(automatika.cas);
				automatika.desiredPressure3[3]:= (automatika.desiredPressure3_previous[3]*(automatika.cas - TIME_TO_INT(TON_0.ET))/automatika.cas) + TIME_TO_INT(TON_0.ET)*(3573)/(automatika.cas);
				automatika.desiredPressure3[4]:= (automatika.desiredPressure3_previous[4]*(automatika.cas - TIME_TO_INT(TON_0.ET))/automatika.cas) + TIME_TO_INT(TON_0.ET)*(3796)/(automatika.cas);
				automatika.desiredPressure3[5]:= (automatika.desiredPressure3_previous[5]*(automatika.cas - TIME_TO_INT(TON_0.ET))/automatika.cas) + TIME_TO_INT(TON_0.ET)*(4104)/(automatika.cas);
				automatika.desiredPressure3[6]:= (automatika.desiredPressure3_previous[6]*(automatika.cas - TIME_TO_INT(TON_0.ET))/automatika.cas) + TIME_TO_INT(TON_0.ET)*(7462)/(automatika.cas);

				automatika.desiredPressureLinear := TIME_TO_INT(TON_0.ET)*10800/((automatika.cas));

				IF TON_0.Q = TRUE THEN
					casovac_start					:= FALSE;
					automatika.step_repeatability	:= 5;
					FOR i:=0 TO 6 BY 1 DO
						automatika.desiredPressure1_previous[i]	:= automatika.desiredPressure1[i];
						automatika.desiredPressure2_previous[i]	:= automatika.desiredPressure2[i];
						automatika.desiredPressure3_previous[i]	:= automatika.desiredPressure3[i];
					END_FOR
				END_IF
			5:	// Pause
				pauza								:= TRUE;
				automatika.step_repeatability		:= 6;
			6:
				IF TON_1.Q = TRUE THEN
					pauza							:= FALSE;
					automatika.step_repeatability	:= 77;
					casovac_start					:= TRUE;
					kameraBool						:= TRUE;
				END_IF
			77:
				IF TON_2.Q = TRUE THEN
					kameraBool						:= FALSE;
					automatika.step_repeatability	:= 7;
				END_IF

			7:	// Point A
				automatika.desiredPressure1[0]:= (automatika.desiredPressure1_previous[0]*(automatika.cas - TIME_TO_INT(TON_0.ET))/automatika.cas) + TIME_TO_INT(TON_0.ET)*(1669)/(automatika.cas);
				automatika.desiredPressure1[1]:= (automatika.desiredPressure1_previous[1]*(automatika.cas - TIME_TO_INT(TON_0.ET))/automatika.cas) + TIME_TO_INT(TON_0.ET)*(3013)/(automatika.cas);
				automatika.desiredPressure1[2]:= (automatika.desiredPressure1_previous[2]*(automatika.cas - TIME_TO_INT(TON_0.ET))/automatika.cas) + TIME_TO_INT(TON_0.ET)*(-4146)/(automatika.cas);
				automatika.desiredPressure1[3]:= (automatika.desiredPressure1_previous[3]*(automatika.cas - TIME_TO_INT(TON_0.ET))/automatika.cas) + TIME_TO_INT(TON_0.ET)*(-8424)/(automatika.cas);
				automatika.desiredPressure1[4]:= (automatika.desiredPressure1_previous[4]*(automatika.cas - TIME_TO_INT(TON_0.ET))/automatika.cas) + TIME_TO_INT(TON_0.ET)*(335)/(automatika.cas);
				automatika.desiredPressure1[5]:= (automatika.desiredPressure1_previous[5]*(automatika.cas - TIME_TO_INT(TON_0.ET))/automatika.cas) + TIME_TO_INT(TON_0.ET)*(2453)/(automatika.cas);
				automatika.desiredPressure1[6]:= (automatika.desiredPressure1_previous[6]*(automatika.cas - TIME_TO_INT(TON_0.ET))/automatika.cas) + TIME_TO_INT(TON_0.ET)*(6053)/(automatika.cas);

				automatika.desiredPressure2[0]:= (automatika.desiredPressure2_previous[0]*(automatika.cas - TIME_TO_INT(TON_0.ET))/automatika.cas) + TIME_TO_INT(TON_0.ET)*(6958)/(automatika.cas);
				automatika.desiredPressure2[1]:= (automatika.desiredPressure2_previous[1]*(automatika.cas - TIME_TO_INT(TON_0.ET))/automatika.cas) + TIME_TO_INT(TON_0.ET)*(4381)/(automatika.cas);
				automatika.desiredPressure2[2]:= (automatika.desiredPressure2_previous[2]*(automatika.cas - TIME_TO_INT(TON_0.ET))/automatika.cas) + TIME_TO_INT(TON_0.ET)*(12008)/(automatika.cas);
				automatika.desiredPressure2[3]:= (automatika.desiredPressure2_previous[3]*(automatika.cas - TIME_TO_INT(TON_0.ET))/automatika.cas) + TIME_TO_INT(TON_0.ET)*(13312)/(automatika.cas);
				automatika.desiredPressure2[4]:= (automatika.desiredPressure2_previous[4]*(automatika.cas - TIME_TO_INT(TON_0.ET))/automatika.cas) + TIME_TO_INT(TON_0.ET)*(8361)/(automatika.cas);
				automatika.desiredPressure2[5]:= (automatika.desiredPressure2_previous[5]*(automatika.cas - TIME_TO_INT(TON_0.ET))/automatika.cas) + TIME_TO_INT(TON_0.ET)*(6761)/(automatika.cas);
				automatika.desiredPressure2[6]:= (automatika.desiredPressure2_previous[6]*(automatika.cas - TIME_TO_INT(TON_0.ET))/automatika.cas) + TIME_TO_INT(TON_0.ET)*(3567)/(automatika.cas);

				automatika.desiredPressure3[0]:= (automatika.desiredPressure3_previous[0]*(automatika.cas - TIME_TO_INT(TON_0.ET))/automatika.cas) + TIME_TO_INT(TON_0.ET)*(4006)/(automatika.cas);
				automatika.desiredPressure3[1]:= (automatika.desiredPressure3_previous[1]*(automatika.cas - TIME_TO_INT(TON_0.ET))/automatika.cas) + TIME_TO_INT(TON_0.ET)*(5379)/(automatika.cas);
				automatika.desiredPressure3[2]:= (automatika.desiredPressure3_previous[2]*(automatika.cas - TIME_TO_INT(TON_0.ET))/automatika.cas) + TIME_TO_INT(TON_0.ET)*(5605)/(automatika.cas);
				automatika.desiredPressure3[3]:= (automatika.desiredPressure3_previous[3]*(automatika.cas - TIME_TO_INT(TON_0.ET))/automatika.cas) + TIME_TO_INT(TON_0.ET)*(3560)/(automatika.cas);
				automatika.desiredPressure3[4]:= (automatika.desiredPressure3_previous[4]*(automatika.cas - TIME_TO_INT(TON_0.ET))/automatika.cas) + TIME_TO_INT(TON_0.ET)*(3900)/(automatika.cas);
				automatika.desiredPressure3[5]:= (automatika.desiredPressure3_previous[5]*(automatika.cas - TIME_TO_INT(TON_0.ET))/automatika.cas) + TIME_TO_INT(TON_0.ET)*(3205)/(automatika.cas);
				automatika.desiredPressure3[6]:= (automatika.desiredPressure3_previous[6]*(automatika.cas - TIME_TO_INT(TON_0.ET))/automatika.cas) + TIME_TO_INT(TON_0.ET)*(2770)/(automatika.cas);

				automatika.desiredPressureLinear := TIME_TO_INT(TON_0.ET)*10800/((automatika.cas));

				IF TON_0.Q = TRUE THEN
					casovac_start					:= FALSE;
					automatika.step_repeatability	:= 8;
					FOR i:=0 TO 6 BY 1 DO
						automatika.desiredPressure1_previous[i]	:= automatika.desiredPressure1[i];
						automatika.desiredPressure2_previous[i]	:= automatika.desiredPressure2[i];
						automatika.desiredPressure3_previous[i]	:= automatika.desiredPressure3[i];
					END_FOR
				END_IF
			8:	// Pause
				pauza								:= TRUE;
				automatika.step_repeatability		:= 9;
			9:
				IF TON_1.Q = TRUE THEN
					pauza							:= FALSE;
					automatika.step_repeatability	:= 99;
					casovac_start					:= TRUE;
					kameraBool						:= TRUE;
				END_IF
			99:
				IF TON_2.Q = TRUE THEN
					kameraBool						:= FALSE;
					automatika.step_repeatability	:= 4;
				END_IF

		END_CASE

	END_IF

END_PROGRAM
```

### Program Logical/meranie (ANSIC, version 1.00.0)

#### global.txt
```
VAR
	    u1 : INT := 0; (**)
	    p1 : REAL := 0; (**)
	    p2 : REAL := 0; (**)
	    p3 : REAL := 0; (**)
	    u2 : INT := 0; (**)
	    result : INT := 0; (**)
END_VAR
```

#### multiword_types.h
```c
/*
 * multiword_types.h
 *
 * Academic License - for use in teaching, academic research, and meeting
 * course requirements at degree granting institutions only.  Not for
 * government, commercial, or other organizational use.
 *
 * Code generation for model "pneutrunkMeranie".
 *
 * Model version              : 1.6
 * Simulink Coder version : 9.8 (R2022b) 13-May-2022
 * C source code generated on : Wed May 24 11:04:27 2023
 *
 * Target selection: bur_grt.tlc
 * Note: GRT includes extra infrastructure and instrumentation for prototyping
 * Embedded hardware selection: Intel->x86/Pentium
 * Code generation objectives: Unspecified
 * Validation result: Not run
 */

#ifndef MULTIWORD_TYPES_H
#define MULTIWORD_TYPES_H
#include "rtwtypes.h"

/*
 * Definitions supporting external data access
 */
typedef int32_T chunk_T;
typedef uint32_T uchunk_T;

/*
 * MultiWord supporting definitions
 */
typedef long int long_T;

/*
 * MultiWord types
 */
typedef struct {
  uint32_T chunks[2];
} int64m_T;

typedef struct {
  int64m_T re;
  int64m_T im;
} cint64m_T;

typedef struct {
  uint32_T chunks[2];
} uint64m_T;

typedef struct {
  uint64m_T re;
  uint64m_T im;
} cuint64m_T;

typedef struct {
  uint32_T chunks[3];
} int96m_T;

typedef struct {
  int96m_T re;
  int96m_T im;
} cint96m_T;

typedef struct {
  uint32_T chunks[3];
} uint96m_T;

typedef struct {
  uint96m_T re;
  uint96m_T im;
} cuint96m_T;

typedef struct {
  uint32_T chunks[4];
} int128m_T;

typedef struct {
  int128m_T re;
  int128m_T im;
} cint128m_T;

typedef struct {
  uint32_T chunks[4];
} uint128m_T;

typedef struct {
  uint128m_T re;
  uint128m_T im;
} cuint128m_T;

typedef struct {
  uint32_T chunks[5];
} int160m_T;

typedef struct {
  int160m_T re;
  int160m_T im;
} cint160m_T;

typedef struct {
  uint32_T chunks[5];
} uint160m_T;

typedef struct {
  uint160m_T re;
  uint160m_T im;
} cuint160m_T;

typedef struct {
  uint32_T chunks[6];
} int192m_T;

typedef struct {
  int192m_T re;
  int192m_T im;
} cint192m_T;

typedef struct {
  uint32_T chunks[6];
} uint192m_T;

typedef struct {
  uint192m_T re;
  uint192m_T im;
} cuint192m_T;

typedef struct {
  uint32_T chunks[7];
} int224m_T;

typedef struct {
  int224m_T re;
  int224m_T im;
} cint224m_T;

typedef struct {
  uint32_T chunks[7];
} uint224m_T;

typedef struct {
  uint224m_T re;
  uint224m_T im;
} cuint224m_T;

typedef struct {
  uint32_T chunks[8];
} int256m_T;

typedef struct {
  int256m_T re;
  int256m_T im;
} cint256m_T;

typedef struct {
  uint32_T chunks[8];
} uint256m_T;

typedef struct {
  uint256m_T re;
  uint256m_T im;
} cuint256m_T;

typedef struct {
  uint32_T chunks[9];
} int288m_T;

typedef struct {
  int288m_T re;
  int288m_T im;
} cint288m_T;

typedef struct {
  uint32_T chunks[9];
} uint288m_T;

typedef struct {
  uint288m_T re;
  uint288m_T im;
} cuint288m_T;

typedef struct {
  uint32_T chunks[10];
} int320m_T;

typedef struct {
  int320m_T re;
  int320m_T im;
} cint320m_T;

typedef struct {
  uint32_T chunks[10];
} uint320m_T;

typedef struct {
  uint320m_T re;
  uint320m_T im;
} cuint320m_T;

typedef struct {
  uint32_T chunks[11];
} int352m_T;

typedef struct {
  int352m_T re;
  int352m_T im;
} cint352m_T;

typedef struct {
  uint32_T chunks[11];
} uint352m_T;

typedef struct {
  uint352m_T re;
  uint352m_T im;
} cuint352m_T;

typedef struct {
  uint32_T chunks[12];
} int384m_T;

typedef struct {
  int384m_T re;
  int384m_T im;
} cint384m_T;

typedef struct {
  uint32_T chunks[12];
} uint384m_T;

typedef struct {
  uint384m_T re;
  uint384m_T im;
} cuint384m_T;

typedef struct {
  uint32_T chunks[13];
} int416m_T;

typedef struct {
  int416m_T re;
  int416m_T im;
} cint416m_T;

typedef struct {
  uint32_T chunks[13];
} uint416m_T;

typedef struct {
  uint416m_T re;
  uint416m_T im;
} cuint416m_T;

typedef struct {
  uint32_T chunks[14];
} int448m_T;

typedef struct {
  int448m_T re;
  int448m_T im;
} cint448m_T;

typedef struct {
  uint32_T chunks[14];
} uint448m_T;

typedef struct {
  uint448m_T re;
  uint448m_T im;
} cuint448m_T;

typedef struct {
  uint32_T chunks[15];
} int480m_T;

typedef struct {
  int480m_T re;
  int480m_T im;
} cint480m_T;

typedef struct {
  uint32_T chunks[15];
} uint480m_T;

typedef struct {
  uint480m_T re;
  uint480m_T im;
} cuint480m_T;

typedef struct {
  uint32_T chunks[16];
} int512m_T;

typedef struct {
  int512m_T re;
  int512m_T im;
} cint512m_T;

typedef struct {
  uint32_T chunks[16];
} uint512m_T;

typedef struct {
  uint512m_T re;
  uint512m_T im;
} cuint512m_T;

typedef struct {
  uint32_T chunks[17];
} int544m_T;

typedef struct {
  int544m_T re;
  int544m_T im;
} cint544m_T;

typedef struct {
  uint32_T chunks[17];
} uint544m_T;

typedef struct {
  uint544m_T re;
  uint544m_T im;
} cuint544m_T;

typedef struct {
  uint32_T chunks[18];
} int576m_T;

typedef struct {
  int576m_T re;
  int576m_T im;
} cint576m_T;

typedef struct {
  uint32_T chunks[18];
} uint576m_T;

typedef struct {
  uint576m_T re;
  uint576m_T im;
} cuint576m_T;

typedef struct {
  uint32_T chunks[19];
} int608m_T;

typedef struct {
  int608m_T re;
  int608m_T im;
} cint608m_T;

typedef struct {
  uint32_T chunks[19];
} uint608m_T;

typedef struct {
  uint608m_T re;
  uint608m_T im;
} cuint608m_T;

typedef struct {
  uint32_T chunks[20];
} int640m_T;

typedef struct {
  int640m_T re;
  int640m_T im;
} cint640m_T;

typedef struct {
  uint32_T chunks[20];
} uint640m_T;

typedef struct {
  uint640m_T re;
  uint640m_T im;
} cuint640m_T;

typedef struct {
  uint32_T chunks[21];
} int672m_T;

typedef struct {
  int672m_T re;
  int672m_T im;
} cint672m_T;

typedef struct {
  uint32_T chunks[21];
} uint672m_T;

typedef struct {
  uint672m_T re;
  uint672m_T im;
} cuint672m_T;

typedef struct {
  uint32_T chunks[22];
} int704m_T;

typedef struct {
  int704m_T re;
  int704m_T im;
} cint704m_T;

typedef struct {
  uint32_T chunks[22];
} uint704m_T;

typedef struct {
  uint704m_T re;
  uint704m_T im;
} cuint704m_T;

typedef struct {
  uint32_T chunks[23];
} int736m_T;

typedef struct {
  int736m_T re;
  int736m_T im;
} cint736m_T;

typedef struct {
  uint32_T chunks[23];
} uint736m_T;

typedef struct {
  uint736m_T re;
  uint736m_T im;
} cuint736m_T;

typedef struct {
  uint32_T chunks[24];
} int768m_T;

typedef struct {
  int768m_T re;
  int768m_T im;
} cint768m_T;

typedef struct {
  uint32_T chunks[24];
} uint768m_T;

typedef struct {
  uint768m_T re;
  uint768m_T im;
} cuint768m_T;

typedef struct {
  uint32_T chunks[25];
} int800m_T;

typedef struct {
  int800m_T re;
  int800m_T im;
} cint800m_T;

typedef struct {
  uint32_T chunks[25];
} uint800m_T;

typedef struct {
  uint800m_T re;
  uint800m_T im;
} cuint800m_T;

typedef struct {
  uint32_T chunks[26];
} int832m_T;

typedef struct {
  int832m_T re;
  int832m_T im;
} cint832m_T;

typedef struct {
  uint32_T chunks[26];
} uint832m_T;

typedef struct {
  uint832m_T re;
  uint832m_T im;
} cuint832m_T;

typedef struct {
  uint32_T chunks[27];
} int864m_T;

typedef struct {
  int864m_T re;
  int864m_T im;
} cint864m_T;

typedef struct {
  uint32_T chunks[27];
} uint864m_T;

typedef struct {
  uint864m_T re;
  uint864m_T im;
} cuint864m_T;

typedef struct {
  uint32_T chunks[28];
} int896m_T;

typedef struct {
  int896m_T re;
  int896m_T im;
} cint896m_T;

typedef struct {
  uint32_T chunks[28];
} uint896m_T;

typedef struct {
  uint896m_T re;
  uint896m_T im;
} cuint896m_T;

typedef struct {
  uint32_T chunks[29];
} int928m_T;

typedef struct {
  int928m_T re;
  int928m_T im;
} cint928m_T;

typedef struct {
  uint32_T chunks[29];
} uint928m_T;

typedef struct {
  uint928m_T re;
  uint928m_T im;
} cuint928m_T;

typedef struct {
  uint32_T chunks[30];
} int960m_T;

typedef struct {
  int960m_T re;
  int960m_T im;
} cint960m_T;

typedef struct {
  uint32_T chunks[30];
} uint960m_T;

typedef struct {
  uint960m_T re;
  uint960m_T im;
} cuint960m_T;

typedef struct {
  uint32_T chunks[31];
} int992m_T;

typedef struct {
  int992m_T re;
  int992m_T im;
} cint992m_T;

typedef struct {
  uint32_T chunks[31];
} uint992m_T;

typedef struct {
  uint992m_T re;
  uint992m_T im;
} cuint992m_T;

typedef struct {
  uint32_T chunks[32];
} int1024m_T;

typedef struct {
  int1024m_T re;
  int1024m_T im;
} cint1024m_T;

typedef struct {
  uint32_T chunks[32];
} uint1024m_T;

typedef struct {
  uint1024m_T re;
  uint1024m_T im;
} cuint1024m_T;

typedef struct {
  uint32_T chunks[33];
} int1056m_T;

typedef struct {
  int1056m_T re;
  int1056m_T im;
} cint1056m_T;

typedef struct {
  uint32_T chunks[33];
} uint1056m_T;

typedef struct {
  uint1056m_T re;
  uint1056m_T im;
} cuint1056m_T;

typedef struct {
  uint32_T chunks[34];
} int1088m_T;

typedef struct {
  int1088m_T re;
  int1088m_T im;
} cint1088m_T;

typedef struct {
  uint32_T chunks[34];
} uint1088m_T;

typedef struct {
  uint1088m_T re;
  uint1088m_T im;
} cuint1088m_T;

typedef struct {
  uint32_T chunks[35];
} int1120m_T;

typedef struct {
  int1120m_T re;
  int1120m_T im;
} cint1120m_T;

typedef struct {
  uint32_T chunks[35];
} uint1120m_T;

typedef struct {
  uint1120m_T re;
  uint1120m_T im;
} cuint1120m_T;

typedef struct {
  uint32_T chunks[36];
} int1152m_T;

typedef struct {
  int1152m_T re;
  int1152m_T im;
} cint1152m_T;

typedef struct {
  uint32_T chunks[36];
} uint1152m_T;

typedef struct {
  uint1152m_T re;
  uint1152m_T im;
} cuint1152m_T;

typedef struct {
  uint32_T chunks[37];
} int1184m_T;

typedef struct {
  int1184m_T re;
  int1184m_T im;
} cint1184m_T;

typedef struct {
  uint32_T chunks[37];
} uint1184m_T;

typedef struct {
  uint1184m_T re;
  uint1184m_T im;
} cuint1184m_T;

typedef struct {
  uint32_T chunks[38];
} int1216m_T;

typedef struct {
  int1216m_T re;
  int1216m_T im;
} cint1216m_T;

typedef struct {
  uint32_T chunks[38];
} uint1216m_T;

typedef struct {
  uint1216m_T re;
  uint1216m_T im;
} cuint1216m_T;

typedef struct {
  uint32_T chunks[39];
} int1248m_T;

typedef struct {
  int1248m_T re;
  int1248m_T im;
} cint1248m_T;

typedef struct {
  uint32_T chunks[39];
} uint1248m_T;

typedef struct {
  uint1248m_T re;
  uint1248m_T im;
} cuint1248m_T;

typedef struct {
  uint32_T chunks[40];
} int1280m_T;

typedef struct {
  int1280m_T re;
  int1280m_T im;
} cint1280m_T;

typedef struct {
  uint32_T chunks[40];
} uint1280m_T;

typedef struct {
  uint1280m_T re;
  uint1280m_T im;
} cuint1280m_T;

typedef struct {
  uint32_T chunks[41];
} int1312m_T;

typedef struct {
  int1312m_T re;
  int1312m_T im;
} cint1312m_T;

typedef struct {
  uint32_T chunks[41];
} uint1312m_T;

typedef struct {
  uint1312m_T re;
  uint1312m_T im;
} cuint1312m_T;

typedef struct {
  uint32_T chunks[42];
} int1344m_T;

typedef struct {
  int1344m_T re;
  int1344m_T im;
} cint1344m_T;

typedef struct {
  uint32_T chunks[42];
} uint1344m_T;

typedef struct {
  uint1344m_T re;
  uint1344m_T im;
} cuint1344m_T;

typedef struct {
  uint32_T chunks[43];
} int1376m_T;

typedef struct {
  int1376m_T re;
  int1376m_T im;
} cint1376m_T;

typedef struct {
  uint32_T chunks[43];
} uint1376m_T;

typedef struct {
  uint1376m_T re;
  uint1376m_T im;
} cuint1376m_T;

typedef struct {
  uint32_T chunks[44];
} int1408m_T;

typedef struct {
  int1408m_T re;
  int1408m_T im;
} cint1408m_T;

typedef struct {
  uint32_T chunks[44];
} uint1408m_T;

typedef struct {
  uint1408m_T re;
  uint1408m_T im;
} cuint1408m_T;

typedef struct {
  uint32_T chunks[45];
} int1440m_T;

typedef struct {
  int1440m_T re;
  int1440m_T im;
} cint1440m_T;

typedef struct {
  uint32_T chunks[45];
} uint1440m_T;

typedef struct {
  uint1440m_T re;
  uint1440m_T im;
} cuint1440m_T;

typedef struct {
  uint32_T chunks[46];
} int1472m_T;

typedef struct {
  int1472m_T re;
  int1472m_T im;
} cint1472m_T;

typedef struct {
  uint32_T chunks[46];
} uint1472m_T;

typedef struct {
  uint1472m_T re;
  uint1472m_T im;
} cuint1472m_T;

typedef struct {
  uint32_T chunks[47];
} int1504m_T;

typedef struct {
  int1504m_T re;
  int1504m_T im;
} cint1504m_T;

typedef struct {
  uint32_T chunks[47];
} uint1504m_T;

typedef struct {
  uint1504m_T re;
  uint1504m_T im;
} cuint1504m_T;

typedef struct {
  uint32_T chunks[48];
} int1536m_T;

typedef struct {
  int1536m_T re;
  int1536m_T im;
} cint1536m_T;

typedef struct {
  uint32_T chunks[48];
} uint1536m_T;

typedef struct {
  uint1536m_T re;
  uint1536m_T im;
} cuint1536m_T;

typedef struct {
  uint32_T chunks[49];
} int1568m_T;

typedef struct {
  int1568m_T re;
  int1568m_T im;
} cint1568m_T;

typedef struct {
  uint32_T chunks[49];
} uint1568m_T;

typedef struct {
  uint1568m_T re;
  uint1568m_T im;
} cuint1568m_T;

typedef struct {
  uint32_T chunks[50];
} int1600m_T;

typedef struct {
  int1600m_T re;
  int1600m_T im;
} cint1600m_T;

typedef struct {
  uint32_T chunks[50];
} uint1600m_T;

typedef struct {
  uint1600m_T re;
  uint1600m_T im;
} cuint1600m_T;

typedef struct {
  uint32_T chunks[51];
} int1632m_T;

typedef struct {
  int1632m_T re;
  int1632m_T im;
} cint1632m_T;

typedef struct {
  uint32_T chunks[51];
} uint1632m_T;

typedef struct {
  uint1632m_T re;
  uint1632m_T im;
} cuint1632m_T;

typedef struct {
  uint32_T chunks[52];
} int1664m_T;

typedef struct {
  int1664m_T re;
  int1664m_T im;
} cint1664m_T;

typedef struct {
  uint32_T chunks[52];
} uint1664m_T;

typedef struct {
  uint1664m_T re;
  uint1664m_T im;
} cuint1664m_T;

typedef struct {
  uint32_T chunks[53];
} int1696m_T;

typedef struct {
  int1696m_T re;
  int1696m_T im;
} cint1696m_T;

typedef struct {
  uint32_T chunks[53];
} uint1696m_T;

typedef struct {
  uint1696m_T re;
  uint1696m_T im;
} cuint1696m_T;

typedef struct {
  uint32_T chunks[54];
} int1728m_T;

typedef struct {
  int1728m_T re;
  int1728m_T im;
} cint1728m_T;

typedef struct {
  uint32_T chunks[54];
} uint1728m_T;

typedef struct {
  uint1728m_T re;
  uint1728m_T im;
} cuint1728m_T;

typedef struct {
  uint32_T chunks[55];
} int1760m_T;

typedef struct {
  int1760m_T re;
  int1760m_T im;
} cint1760m_T;

typedef struct {
  uint32_T chunks[55];
} uint1760m_T;

typedef struct {
  uint1760m_T re;
  uint1760m_T im;
} cuint1760m_T;

typedef struct {
  uint32_T chunks[56];
} int1792m_T;

typedef struct {
  int1792m_T re;
  int1792m_T im;
} cint1792m_T;

typedef struct {
  uint32_T chunks[56];
} uint1792m_T;

typedef struct {
  uint1792m_T re;
  uint1792m_T im;
} cuint1792m_T;

typedef struct {
  uint32_T chunks[57];
} int1824m_T;

typedef struct {
  int1824m_T re;
  int1824m_T im;
} cint1824m_T;

typedef struct {
  uint32_T chunks[57];
} uint1824m_T;

typedef struct {
  uint1824m_T re;
  uint1824m_T im;
} cuint1824m_T;

typedef struct {
  uint32_T chunks[58];
} int1856m_T;

typedef struct {
  int1856m_T re;
  int1856m_T im;
} cint1856m_T;

typedef struct {
  uint32_T chunks[58];
} uint1856m_T;

typedef struct {
  uint1856m_T re;
  uint1856m_T im;
} cuint1856m_T;

typedef struct {
  uint32_T chunks[59];
} int1888m_T;

typedef struct {
  int1888m_T re;
  int1888m_T im;
} cint1888m_T;

typedef struct {
  uint32_T chunks[59];
} uint1888m_T;

typedef struct {
  uint1888m_T re;
  uint1888m_T im;
} cuint1888m_T;

typedef struct {
  uint32_T chunks[60];
} int1920m_T;

typedef struct {
  int1920m_T re;
  int1920m_T im;
} cint1920m_T;

typedef struct {
  uint32_T chunks[60];
} uint1920m_T;

typedef struct {
  uint1920m_T re;
  uint1920m_T im;
} cuint1920m_T;

typedef struct {
  uint32_T chunks[61];
} int1952m_T;

typedef struct {
  int1952m_T re;
  int1952m_T im;
} cint1952m_T;

typedef struct {
  uint32_T chunks[61];
} uint1952m_T;

typedef struct {
  uint1952m_T re;
  uint1952m_T im;
} cuint1952m_T;

typedef struct {
  uint32_T chunks[62];
} int1984m_T;

typedef struct {
  int1984m_T re;
  int1984m_T im;
} cint1984m_T;

typedef struct {
  uint32_T chunks[62];
} uint1984m_T;

typedef struct {
  uint1984m_T re;
  uint1984m_T im;
} cuint1984m_T;

typedef struct {
  uint32_T chunks[63];
} int2016m_T;

typedef struct {
  int2016m_T re;
  int2016m_T im;
} cint2016m_T;

typedef struct {
  uint32_T chunks[63];
} uint2016m_T;

typedef struct {
  uint2016m_T re;
  uint2016m_T im;
} cuint2016m_T;

typedef struct {
  uint32_T chunks[64];
} int2048m_T;

typedef struct {
  int2048m_T re;
  int2048m_T im;
} cint2048m_T;

typedef struct {
  uint32_T chunks[64];
} uint2048m_T;

typedef struct {
  uint2048m_T re;
  uint2048m_T im;
} cuint2048m_T;

#endif                                 /* MULTIWORD_TYPES_H */
```

#### pneutrunkMeranie.c
```c
/*
 * pneutrunkMeranie.c
 *
 * Academic License - for use in teaching, academic research, and meeting
 * course requirements at degree granting institutions only.  Not for
 * government, commercial, or other organizational use.
 *
 * Code generation for model "pneutrunkMeranie".
 *
 * Model version              : 1.6
 * Simulink Coder version : 9.8 (R2022b) 13-May-2022
 * C source code generated on : Wed May 24 11:04:27 2023
 *
 * Target selection: bur_grt.tlc
 * Note: GRT includes extra infrastructure and instrumentation for prototyping
 * Embedded hardware selection: Intel->x86/Pentium
 * Code generation objectives: Unspecified
 * Validation result: Not run
 */

#include "pneutrunkMeranie.h"
#include <string.h>
#include "rt_nonfinite.h"
#include "pneutrunkMeranie_dt.h"

/* Block signals (default storage) */
B_pneutrunkMeranie_T pneutrunkMeranie_B;

/* Block states (default storage) */
DW_pneutrunkMeranie_T pneutrunkMeranie_DW;

/* Real-time model */
static RT_MODEL_pneutrunkMeranie_T pneutrunkMeranie_M_;
RT_MODEL_pneutrunkMeranie_T *const pneutrunkMeranie_M = &pneutrunkMeranie_M_;

/* Model output function */
void pneutrunkMeranie_output(void)
{
  /* S-Function (bur_in): '<Root>/Input3' */
  pneutrunkMeranie_B.Input3 = u1;

  /* S-Function (bur_in): '<Root>/Input' */
  pneutrunkMeranie_B.Input = p1;

  /* S-Function (bur_in): '<Root>/Input1' */
  pneutrunkMeranie_B.Input1 = p2;

  /* S-Function (bur_in): '<Root>/Input2' */
  pneutrunkMeranie_B.Input2 = p3;

  /* S-Function (bur_in): '<Root>/Input4' */
  pneutrunkMeranie_B.Input4 = u2;

  /* S-Function (bur_in): '<Root>/Input5' */
  pneutrunkMeranie_B.Input5 = result;
}

/* Model update function */
void pneutrunkMeranie_update(void)
{
  /* Update absolute time for base rate */
  /* The "clockTick0" counts the number of times the code of this task has
   * been executed. The absolute time is the multiplication of "clockTick0"
   * and "Timing.stepSize0". Size of "clockTick0" ensures timer will not
   * overflow during the application lifespan selected.
   * Timer of this task consists of two 32 bit unsigned integers.
   * The two integers represent the low bits Timing.clockTick0 and the high bits
   * Timing.clockTickH0. When the low bit overflows to 0, the high bits increment.
   */
  if (!(++pneutrunkMeranie_M->Timing.clockTick0)) {
    ++pneutrunkMeranie_M->Timing.clockTickH0;
  }

  pneutrunkMeranie_M->Timing.t[0] = pneutrunkMeranie_M->Timing.clockTick0 *
    pneutrunkMeranie_M->Timing.stepSize0 +
    pneutrunkMeranie_M->Timing.clockTickH0 *
    pneutrunkMeranie_M->Timing.stepSize0 * 4294967296.0;
}

/* Model initialize function */
void pneutrunkMeranie_initialize(void)
{
}

/* Model terminate function */
void pneutrunkMeranie_terminate(void)
{
  /* (no terminate code required) */
}

/*========================================================================*
 * Start of Classic call interface                                        *
 *========================================================================*/
void MdlOutputs(int_T tid)
{
  pneutrunkMeranie_output();
  UNUSED_PARAMETER(tid);
}

void MdlUpdate(int_T tid)
{
  pneutrunkMeranie_update();
  UNUSED_PARAMETER(tid);
}

void MdlInitializeSizes(void)
{
}

void MdlInitializeSampleTimes(void)
{
}

void MdlInitialize(void)
{
}

void MdlStart(void)
{
  pneutrunkMeranie_initialize();
}

void MdlTerminate(void)
{
  pneutrunkMeranie_terminate();
}

/* Registration function */
RT_MODEL_pneutrunkMeranie_T *pneutrunkMeranie(void)
{
  /* Registration code */

  /* initialize non-finites */
  rt_InitInfAndNaN(sizeof(real_T));

  /* initialize real-time model */
  (void) memset((void *)pneutrunkMeranie_M, 0,
                sizeof(RT_MODEL_pneutrunkMeranie_T));

  /* Initialize timing info */
  {
    int_T *mdlTsMap = pneutrunkMeranie_M->Timing.sampleTimeTaskIDArray;
    mdlTsMap[0] = 0;

    /* polyspace +2 MISRA2012:D4.1 [Justified:Low] "pneutrunkMeranie_M points to
       static memory which is guaranteed to be non-NULL" */
    pneutrunkMeranie_M->Timing.sampleTimeTaskIDPtr = (&mdlTsMap[0]);
    pneutrunkMeranie_M->Timing.sampleTimes =
      (&pneutrunkMeranie_M->Timing.sampleTimesArray[0]);
    pneutrunkMeranie_M->Timing.offsetTimes =
      (&pneutrunkMeranie_M->Timing.offsetTimesArray[0]);

    /* task periods */
    pneutrunkMeranie_M->Timing.sampleTimes[0] = (0.1);

    /* task offsets */
    pneutrunkMeranie_M->Timing.offsetTimes[0] = (0.0);
  }

  rtmSetTPtr(pneutrunkMeranie_M, &pneutrunkMeranie_M->Timing.tArray[0]);

  {
    int_T *mdlSampleHits = pneutrunkMeranie_M->Timing.sampleHitArray;
    mdlSampleHits[0] = 1;
    pneutrunkMeranie_M->Timing.sampleHits = (&mdlSampleHits[0]);
  }

  rtmSetTFinal(pneutrunkMeranie_M, -1);
  pneutrunkMeranie_M->Timing.stepSize0 = 0.1;

  /* External mode info */
  pneutrunkMeranie_M->Sizes.checksums[0] = (272960474U);
  pneutrunkMeranie_M->Sizes.checksums[1] = (2602910742U);
  pneutrunkMeranie_M->Sizes.checksums[2] = (2322055424U);
  pneutrunkMeranie_M->Sizes.checksums[3] = (1324330691U);

  {
    static const sysRanDType rtAlwaysEnabled = SUBSYS_RAN_BC_ENABLE;
    static RTWExtModeInfo rt_ExtModeInfo;
    static const sysRanDType *systemRan[1];
    pneutrunkMeranie_M->extModeInfo = (&rt_ExtModeInfo);
    rteiSetSubSystemActiveVectorAddresses(&rt_ExtModeInfo, systemRan);
    systemRan[0] = &rtAlwaysEnabled;
    rteiSetModelMappingInfoPtr(pneutrunkMeranie_M->extModeInfo,
      &pneutrunkMeranie_M->SpecialInfo.mappingInfo);
    rteiSetChecksumsPtr(pneutrunkMeranie_M->extModeInfo,
                        pneutrunkMeranie_M->Sizes.checksums);
    rteiSetTPtr(pneutrunkMeranie_M->extModeInfo, rtmGetTPtr(pneutrunkMeranie_M));
  }

  pneutrunkMeranie_M->solverInfoPtr = (&pneutrunkMeranie_M->solverInfo);
  pneutrunkMeranie_M->Timing.stepSize = (0.1);
  rtsiSetFixedStepSize(&pneutrunkMeranie_M->solverInfo, 0.1);
  rtsiSetSolverMode(&pneutrunkMeranie_M->solverInfo, SOLVER_MODE_SINGLETASKING);

  /* block I/O */
  pneutrunkMeranie_M->blockIO = ((void *) &pneutrunkMeranie_B);
  (void) memset(((void *) &pneutrunkMeranie_B), 0,
                sizeof(B_pneutrunkMeranie_T));

  {
    pneutrunkMeranie_B.Input = 0.0F;
    pneutrunkMeranie_B.Input1 = 0.0F;
    pneutrunkMeranie_B.Input2 = 0.0F;
  }

  /* states (dwork) */
  pneutrunkMeranie_M->dwork = ((void *) &pneutrunkMeranie_DW);
  (void) memset((void *)&pneutrunkMeranie_DW, 0,
                sizeof(DW_pneutrunkMeranie_T));

  /* data type transition information */
  {
    static DataTypeTransInfo dtInfo;
    (void) memset((char_T *) &dtInfo, 0,
                  sizeof(dtInfo));
    pneutrunkMeranie_M->SpecialInfo.mappingInfo = (&dtInfo);
    dtInfo.numDataTypes = 19;
    dtInfo.dataTypeSizes = &rtDataTypeSizes[0];
    dtInfo.dataTypeNames = &rtDataTypeNames[0];

    /* Block I/O transition table */
    dtInfo.BTransTable = &rtBTransTable;
  }

  /* Initialize Sizes */
  pneutrunkMeranie_M->Sizes.numContStates = (0);/* Number of continuous states */
  pneutrunkMeranie_M->Sizes.numY = (0);/* Number of model outputs */
  pneutrunkMeranie_M->Sizes.numU = (0);/* Number of model inputs */
  pneutrunkMeranie_M->Sizes.sysDirFeedThru = (0);/* The model is not direct feedthrough */
  pneutrunkMeranie_M->Sizes.numSampTimes = (1);/* Number of sample times */
  pneutrunkMeranie_M->Sizes.numBlocks = (14);/* Number of blocks */
  pneutrunkMeranie_M->Sizes.numBlockIO = (6);/* Number of block outputs */
  return pneutrunkMeranie_M;
}

/*========================================================================*
 * End of Classic call interface                                          *
 *========================================================================*/
```


### Program Logical/solo_reg

#### rtmodel.h
```c
/*
 *  rtmodel.h:
 *
 * Academic License - for use in teaching, academic research, and meeting
 * course requirements at degree granting institutions only.  Not for
 * government, commercial, or other organizational use.
 *
 * Code generation for model "pneutr2_reg_FF_stiff".
 *
 * Model version              : 4.30
 * Simulink Coder version : 9.9 (R2023a) 19-Nov-2022
 * C source code generated on : Thu Feb 15 10:44:02 2024
 *
 * Target selection: bur_grt.tlc
 * Note: GRT includes extra infrastructure and instrumentation for prototyping
 * Embedded hardware selection: Intel->x86/Pentium
 * Code generation objectives: Unspecified
 * Validation result: Not run
 */

#ifndef RTW_HEADER_rtmodel_h_
#define RTW_HEADER_rtmodel_h_
#include "pneutr2_reg_FF_stiff.h"
#define GRTINTERFACE                   1
#endif                                 /* RTW_HEADER_rtmodel_h_ */
```

#### zero_crossing_types.h
```c
/*
 * zero_crossing_types.h
 *
 * Academic License - for use in teaching, academic research, and meeting
 * course requirements at degree granting institutions only.  Not for
 * government, commercial, or other organizational use.
 *
 * Code generation for model "pneutr2_reg_FF_stiff".
 *
 * Model version              : 4.30
 * Simulink Coder version : 9.9 (R2023a) 19-Nov-2022
 * C source code generated on : Thu Feb 15 10:44:02 2024
 *
 * Target selection: bur_grt.tlc
 * Note: GRT includes extra infrastructure and instrumentation for prototyping
 * Embedded hardware selection: Intel->x86/Pentium
 * Code generation objectives: Unspecified
 * Validation result: Not run
 */

#ifndef ZERO_CROSSING_TYPES_H
#define ZERO_CROSSING_TYPES_H
#include "rtwtypes.h"

/* Trigger directions: falling, either, and rising */
typedef enum {
  FALLING_ZERO_CROSSING = -1,
  ANY_ZERO_CROSSING = 0,
  RISING_ZERO_CROSSING = 1
} ZCDirection;

/* Previous state of a trigger signal */
typedef uint8_T ZCSigState;

/* Initial value of a trigger zero crossing signal */
#define UNINITIALIZED_ZCSIG            0x03U
#define NEG_ZCSIG                      0x02U
#define POS_ZCSIG                      0x01U
#define ZERO_ZCSIG                     0x00U

/* Current state of a trigger signal */
typedef enum { FALLING_ZCEVENT = -1, NO_ZCEVENT = 0, RISING_ZCEVENT = 1 }
  ZCEventType;

#endif                                 /* ZERO_CROSSING_TYPES_H */
```
